// TIA Portal project "CEPS-输送线" (V14)

(* hardware
DEVICE "S7-1200 station_1"  S7-1200 Station
   slot 0: "Rack_0"  S7-1200 Rack  Rack  V1.0
   slot 1: "CEPS传输线"  CPU 1214C DC/DC/DC  6ES7 214-1AG40-0XB0  V4.2
   slot 2: "DI 16x24VDC/DQ 16xRelay_1"  SM 1223 DI16/DQ16 x relay  6ES7 223-1PL32-0XB0  V2.0
   slot 3: "AQ 2x14BIT_1"  SM 1232 AQ2  6ES7 232-4HB32-0XB0  V2.0
DEVICE "HMI"  KTP900 Basic PN
   slot 0: "KTP900 Basic PN"  KTP900 Basic PN  6AV2 123-2JB03-0AX0  14.0.1.0
   slot 1: "HMI_RT_2"  KTP900 Basic PN  6AV2 123-2JB03-0AX0  14.0.1.0
   slot 5: "HMI.IE_CP_1"  PROFINET Interface  14.0.1.0
      slot 1: "PROFINET Interface_1"  PROFINET Interface
         slot 1: "Port_1"  Port
*)

// ===== PLC "CEPS传输线"  CPU 1214C DC/DC/DC =====

VAR_GLOBAL   // PLC tag table "默认变量表"
   "前/后急停按钮" AT %I0.0 : Bool;
   "前/后启动按钮" AT %I0.1 : Bool;
   "前输送线电机变频器报警" AT %I0.2 : Bool;
   "后输送线电机变频器报警" AT %I0.3 : Bool;
   "后方下轨道进料口有料检测" AT %I0.4 : Bool;
   "后升降台有料检测" AT %I0.5 : Bool;
   "前方下轨道出料口有料检测" AT %I0.6 : Bool;
   "前升降台有料检测" AT %I0.7 : Bool;
   "备用2" AT %I1.0 : Bool;
   "前升降台升到位" AT %I1.1 : Bool;
   "前升降台降到位" AT %I1.2 : Bool;
   "后升降台升到位" AT %I1.3 : Bool;
   "后升降台降到位" AT %I1.4 : Bool;
   "备用1" AT %I1.5 : Bool;
   "工位1放行按钮" AT %I2.0 : Bool;
   "工位2放行按钮" AT %I2.1 : Bool;
   "工位3放行按钮" AT %I2.2 : Bool;
   "工位4放行按钮" AT %I2.3 : Bool;
   "工位5放行按钮" AT %I2.4 : Bool;
   "工位6放行按钮" AT %I2.5 : Bool;
   "工位7放行按钮" AT %I2.6 : Bool;
   "前升降台上轨道进料口料盘有料防呆检测" AT %I2.7 : Bool;
   "工位1光电检测" AT %I3.0 : Bool;
   "工位2光电检测" AT %I3.1 : Bool;
   "工位3光电检测" AT %I3.2 : Bool;
   "工位4光电检测" AT %I3.3 : Bool;
   "工位5光电检测" AT %I3.4 : Bool;
   "工位6光电检测" AT %I3.5 : Bool;
   "工位7光电检测" AT %I3.6 : Bool;
   "备用3" AT %I3.7 : Bool;
   "前输送电机启动" AT %Q0.0 : Bool;
   "前输送电机故障复位" AT %Q0.1 : Bool;
   "后输送电机启动" AT %Q0.2 : Bool;
   "后输送电机故障复位" AT %Q0.3 : Bool;
   "前升降台电机正转" AT %Q0.4 : Bool;
   "前升降台电机反转" AT %Q0.5 : Bool;
   "后升降台电机正转" AT %Q0.6 : Bool;
   "后升降台电机反转" AT %Q0.7 : Bool;
   "总气源控制" AT %Q1.0 : Bool;
   "工位3阻挡气缸上升" AT %Q1.1 : Bool;
   "工位1阻挡气缸下降" AT %Q2.0 : Bool;
   "工位2阻挡气缸下降" AT %Q2.1 : Bool;
   "工位3阻挡气缸下降" AT %Q2.2 : Bool;
   "工位4阻挡气缸下降" AT %Q2.3 : Bool;
   "工位5阻挡气缸下降" AT %Q2.4 : Bool;
   "工位6阻挡气缸下降" AT %Q2.5 : Bool;
   "工位7阻挡气缸下降" AT %Q2.6 : Bool;
   "后方下轨道进料口阻挡气缸下降" AT %Q2.7 : Bool;
   "前升降气缸上升" AT %Q3.0 : Bool;
   "前升降气缸下降" AT %Q3.1 : Bool;
   "后升降气缸上升" AT %Q3.2 : Bool;
   "后升降气缸下降" AT %Q3.3 : Bool;
   "后方下轨道阻挡气缸下降" AT %Q3.4 : Bool;
   "后方下轨道阻挡气缸上升" AT %Q3.5 : Bool;
   "工位4阻挡气缸上升" AT %Q3.6 : Bool;
   "工位5阻挡气缸上升" AT %Q3.7 : Bool;
   "System_Byte" AT %MB1 : Byte;
   "FirstScan" AT %M1.0 : Bool;
   "DiagStatusUpdate" AT %M1.1 : Bool;
   "AlwaysTRUE" AT %M1.2 : Bool;
   "AlwaysFALSE" AT %M1.3 : Bool;
   "Clock_Byte" AT %MB0 : Byte;
   "Clock_10Hz" AT %M0.0 : Bool;
   "Clock_5Hz" AT %M0.1 : Bool;
   "Clock_2.5Hz" AT %M0.2 : Bool;
   "Clock_2Hz" AT %M0.3 : Bool;
   "Clock_1.25Hz" AT %M0.4 : Bool;
   "Clock_1Hz" AT %M0.5 : Bool;
   "Clock_0.625Hz" AT %M0.6 : Bool;
   "Clock_0.5Hz" AT %M0.7 : Bool;
   "前输送线电机启动HMI" AT %M10.0 : Bool;
   "前输送线电机停止HMI" AT %M10.1 : Bool;
   "后输送线电机启动HMI" AT %M10.2 : Bool;
   "后输送线电机停止HMI" AT %M10.3 : Bool;
   "前升降台内部电机正转HMI" AT %M10.4 : Bool;
   "前升降台内部电机反转HMI" AT %M10.5 : Bool;
   "前升降台内部电机停止运行HMI" AT %M10.6 : Bool;
   "后升降台内部电机正转HMI" AT %M10.7 : Bool;
   "后升降台内部电机反转HMI" AT %M11.0 : Bool;
   "后升降台内部电机停止运行HMI" AT %M11.1 : Bool;
   "前升降气缸上升HMI" AT %M11.2 : Bool;
   "前升降气缸下降HMI" AT %M11.3 : Bool;
   "后升降气缸上升HMI" AT %M11.4 : Bool;
   "后升降气缸下降HMI" AT %M11.5 : Bool;
   "工位1阻挡气缸上升HMI" AT %M11.6 : Bool;
   "工位1阻挡气缸下降HMI" AT %M11.7 : Bool;
   "工位2阻挡气缸上升HMI" AT %M12.0 : Bool;
   "工位2阻挡气缸下降HMI" AT %M12.1 : Bool;
   "工位3阻挡气缸上升HMI" AT %M12.2 : Bool;
   "工位3阻挡气缸下降HMI" AT %M12.3 : Bool;
   "工位4阻挡气缸上升HMI" AT %M12.4 : Bool;
   "工位4阻挡气缸下降HMI" AT %M12.5 : Bool;
   "工位5阻挡气缸上升HMI" AT %M12.6 : Bool;
   "工位5阻挡气缸下降HMI" AT %M12.7 : Bool;
   "Tag_1" AT %Q4.0 : Bool;
   "工位6阻挡气缸上升HMI" AT %M13.0 : Bool;
   "工位6阻挡气缸下降HMI" AT %M13.1 : Bool;
   "工位7阻挡气缸上升HMI" AT %M13.2 : Bool;
   "工位7阻挡气缸下降HMI" AT %M13.3 : Bool;
   "后方下轨道进料口阻挡气缸上升HMI" AT %M13.4 : Bool;
   "后方下轨道进料口阻挡气缸下降HMI" AT %M13.5 : Bool;
   "后方下轨道阻挡气缸上升HMI" AT %M13.6 : Bool;
   "后方下轨道阻挡气缸下降HMI" AT %M13.7 : Bool;
   "Auto_step" AT %MW50 : Int;
   "Tag_3" AT %MW52 : Int;
   "线体启动HMI" AT %M20.0 : Bool;
   "P0" AT %M4000.0 : Bool;
   "P1" AT %M4000.1 : Bool;
   "P2" AT %M4000.2 : Bool;
   "P3" AT %M4000.3 : Bool;
   "P4" AT %M4000.4 : Bool;
   "P5" AT %M4000.5 : Bool;
   "P6" AT %M4000.6 : Bool;
   "P7" AT %M4000.7 : Bool;
   "P8" AT %M4001.0 : Bool;
   "P9" AT %M4001.1 : Bool;
   "P10" AT %M4001.2 : Bool;
   "P11" AT %M4001.3 : Bool;
   "P12" AT %M4001.4 : Bool;
   "P13" AT %M4001.5 : Bool;
   "P14" AT %M4001.6 : Bool;
   "P15" AT %M4001.7 : Bool;
   "P16" AT %M4002.0 : Bool;
   "P17" AT %M4002.1 : Bool;
   "P18" AT %M4002.2 : Bool;
   "P19" AT %M4002.3 : Bool;
   "P20" AT %M4002.4 : Bool;
   "P21" AT %M4002.5 : Bool;
   "P22" AT %M4002.6 : Bool;
   "P23" AT %M4002.7 : Bool;
   "P24" AT %M4003.0 : Bool;
   "P25" AT %M4003.1 : Bool;
   "P26" AT %M4003.2 : Bool;
   "P27" AT %M4003.3 : Bool;
   "P28" AT %M4003.4 : Bool;
   "P29" AT %M4003.5 : Bool;
   "P30" AT %M4003.6 : Bool;
   "P31" AT %M4003.7 : Bool;
   "P32" AT %M4004.0 : Bool;
   "P33" AT %M4004.1 : Bool;
   "P34" AT %M4004.2 : Bool;
   "P35" AT %M4004.3 : Bool;
   "P36" AT %M4004.4 : Bool;
   "P37" AT %M4004.5 : Bool;
   "P38" AT %M4004.6 : Bool;
   "P39" AT %M4004.7 : Bool;
   "P40" AT %M4005.0 : Bool;
   "P41" AT %M4005.1 : Bool;
   "P42" AT %M4005.2 : Bool;
   "P43" AT %M4005.3 : Bool;
   "P44" AT %M4005.4 : Bool;
   "P45" AT %M4005.5 : Bool;
   "P46" AT %M4005.6 : Bool;
   "P47" AT %M4005.7 : Bool;
   "P48" AT %M4006.0 : Bool;
   "P49" AT %M4006.1 : Bool;
   "P50" AT %M4006.2 : Bool;
   "P51" AT %M4006.3 : Bool;
   "P52" AT %M4006.4 : Bool;
   "P53" AT %M4006.5 : Bool;
   "P54" AT %M4006.6 : Bool;
   "P55" AT %M4006.7 : Bool;
   "P56" AT %M4007.0 : Bool;
   "P57" AT %M4007.1 : Bool;
   "P58" AT %M4007.2 : Bool;
   "P59" AT %M4007.3 : Bool;
   "P60" AT %M4007.4 : Bool;
   "P61" AT %M4007.5 : Bool;
   "P62" AT %M4007.6 : Bool;
   "P63" AT %M4007.7 : Bool;
   "P64" AT %M4008.0 : Bool;
   "P65" AT %M4008.1 : Bool;
   "P66" AT %M4008.2 : Bool;
   "P67" AT %M4008.3 : Bool;
   "P68" AT %M4008.4 : Bool;
   "P69" AT %M4008.5 : Bool;
   "P70" AT %M4008.6 : Bool;
   "P71" AT %M4008.7 : Bool;
   "P72" AT %M4009.0 : Bool;
   "P73" AT %M4009.1 : Bool;
   "P74" AT %M4009.2 : Bool;
   "P75" AT %M4009.3 : Bool;
   "P76" AT %M4009.4 : Bool;
   "P77" AT %M4009.5 : Bool;
   "P78" AT %M4009.6 : Bool;
   "P79" AT %M4009.7 : Bool;
   "P80" AT %M4010.0 : Bool;
   "P81" AT %M4010.1 : Bool;
   "P82" AT %M4010.2 : Bool;
   "P83" AT %M4010.3 : Bool;
   "P84" AT %M4010.4 : Bool;
   "P85" AT %M4010.5 : Bool;
   "P86" AT %M4010.6 : Bool;
   "P87" AT %M4010.7 : Bool;
   "P88" AT %M4011.0 : Bool;
   "P89" AT %M4011.1 : Bool;
   "P90" AT %M4011.2 : Bool;
   "P91" AT %M4011.3 : Bool;
   "P92" AT %M4011.4 : Bool;
   "P93" AT %M4011.5 : Bool;
   "P94" AT %M4011.6 : Bool;
   "P95" AT %M4011.7 : Bool;
   "P96" AT %M4012.0 : Bool;
   "P97" AT %M4012.1 : Bool;
   "P98" AT %M4012.2 : Bool;
   "P99" AT %M4012.3 : Bool;
   "P100" AT %M4012.4 : Bool;
   "线体停止HMI" AT %M20.1 : Bool;
   "前升降台皮带电机正在工作" AT %M100.0 : Bool;
   "后升降台皮带电机正在工作" AT %M100.1 : Bool;
   "前升降台皮带电机显示到HMI状态号" AT %MW2000 : Word;
   "Tag_2" AT %QW112 : Int;
   "Tag_4" AT %QW114 : Int;
   "后升降台皮带电机显示到HMI状态号" AT %MW2002 : Int;
   "前输送线电机显示到HMI状态号" AT %MW2004 : Int;
   "后输送线电机显示到HMI状态号" AT %MW2006 : Int;
   "故障复位HMI" AT %M20.2 : Bool;
   "前升降气缸上升超时报警" AT %M1000.0 : Bool;
   "前升降气缸下降超时报警" AT %M1000.1 : Bool;
   "报警1" AT %MW1000 : Int;
   "后升降气缸上升超时报警" AT %M1000.2 : Bool;
   "后升降气缸下降超时报警" AT %M1000.3 : Bool;
   "前输送电机变频器故障报警" AT %M1000.4 : Bool;
   "后输送电机变频器故障报警" AT %M1000.5 : Bool;
   "急停按下报警" AT %M1000.6 : Bool;
   "设备状态号" AT %MW54 : Int;
   "工位7按钮已按下，待工件流入前升降台，禁止工位7按钮触发" AT %M100.2 : Bool;
   "放行判断" AT %M100.3 : Bool;
END_VAR

DATA_BLOCK "MB_TCON"   // DB1
{ S7_Optimized_Access := 'TRUE' }
VERSION : 0.1
   VAR
      MB_TCON : TCON_IP_v4;
   END_VAR
BEGIN
   MB_TCON.InterfaceId := 64;
   MB_TCON.ID := 1;
   MB_TCON.LocalPort := 502;
END_DATA_BLOCK

DATA_BLOCK "保持数据块"   // DB23
{ S7_Optimized_Access := 'FALSE' }
VERSION : 0.1
   VAR
      产品型号 : Int;
      前输送电机变频器设定频率 : Int;
      后输送电机变频器设定频率 : Int;
      "手动放行/自动放行" : Bool;
      滑移力检测工位 : Int;
      上柱管轴承压装工位 : Int;
      拉轴工位 : Int;
      手柄装配工位 : Int;
      上下柱管压装工位 : Int;
      滑移力复测工位 : Int;
      手柄调节机构工位 : Int;
   END_VAR
BEGIN
END_DATA_BLOCK

DATA_BLOCK "MB_DATA"   // DB100
{ S7_Optimized_Access := 'FALSE' }
VERSION : 0.1
   VAR
      设备编号 : Int := 0;
      产品型号 : Int := 0;
      设备状态 : Int;
      错误代码 : Int := 0;
      当前曲线 : Int := 0;
      工位1状态 : Int := 0;
      工位2状态 : Int;
      工位3状态 : Int;
      工位1生产结果 : Int;
      工位2生产结果 : Int;
      工位3生产结果 : Int;
      备用_1 : Int;
      备用_2 : Int;
      备用_3 : Int;
      备用_4 : Int;
      备用_5 : Int;
      复测拉压力传感器 : Array[0..4] of Real;
      复测位移传感器 : Array[0..4] of Real;
      拉轴拉压力传感器 : Array[0..4] of Real;
      传感器4 : Array[0..4] of Real;
      传感器5 : Array[0..4] of Real;
      传感器6 : Array[0..4] of Real;
      传感器7 : Array[0..4] of Real;
      传感器8 : Array[0..4] of Real;
      传感器9 : Array[0..4] of Real;
      传感器10 : Array[0..4] of Real;
      传感器11 : Array[0..4] of Real;
      传感器12 : Array[0..4] of Real;
      传感器13 : Array[0..4] of Real;
      传感器14 : Array[0..4] of Real;
   END_VAR
BEGIN
   复测拉压力传感器[0] := 0.0;   // 压力值
   复测拉压力传感器[1] := 0.0;
   复测位移传感器[0] := 0.0;   // 位移值
   复测位移传感器[1] := 0.0;
   拉轴拉压力传感器[0] := 0.0;   // 压力值
   拉轴拉压力传感器[1] := 0.0;
   复测拉压力传感器[2] := 0.0;
   复测拉压力传感器[3] := 0.0;
   复测拉压力传感器[4] := 0.0;
   复测位移传感器[2] := 0.0;
   复测位移传感器[3] := 0.0;
   复测位移传感器[4] := 0.0;
   拉轴拉压力传感器[2] := 0.0;
   拉轴拉压力传感器[3] := 0.0;
   拉轴拉压力传感器[4] := 0.0;
   传感器6[0] := 0.0;   // 输入轴角度
   传感器6[1] := 0.0;   // 输出轴角度
   传感器6[2] := 0.0;   // 流量
   传感器6[3] := 0.0;   // 输入轴位移
   传感器6[4] := 0.0;
   传感器4[0] := 0.0;   // 量程下限
   传感器4[1] := 200.0;   // 量程上限
   传感器4[2] := 0.0;   // 原始值
   传感器4[3] := 0.0;   // 偏移值
   传感器4[4] := 0.0;   // 标定值
   传感器5[4] := 0.0;   // 标定值
   传感器5[3] := 0.0;   // 偏移值
   传感器5[2] := 0.0;   // 原始值
   传感器5[1] := 2.5;   // 量程上限
   传感器5[0] := 0.0;   // 量程下限
   传感器8[4] := 65.0;   // 温度上限
   传感器8[3] := 35.0;   // 温度下限
   // 传感器9[0] : 接近距离
   // 传感器9[1] : 接近速度
   // 传感器9[2] : 套入距离
   // 传感器9[3] : 套入速度
   // 传感器10[1] : 摆动角度
   // 传感器10[2] : 摆动速度
   // 传感器10[0] : 状态
   // 传感器10[3] : 保护扭矩
   // 传感器12[0] : 速度
   // 传感器12[1] : 换向扭矩
   // 传感器8[0] : 系统流量
   // 传感器8[1] : 试验流量
   // 传感器8[2] : 试验压力
   // 传感器7[0] : 输入轴角度下限
   // 传感器7[1] : 输入轴角度上限
   // 传感器7[2] : 输出轴角度下限
   // 传感器7[3] : 输出轴角度上限
   // 传感器7[4] : 总圈数
   // 传感器13[0] : 内泄露时间
   // 传感器11[0] : 状态
   // 传感器11[1] : 摆动角度
   // 传感器11[2] : 摆动速度
   // 传感器11[3] : 保护扭矩
   // 传感器14[0] : 输入轴速度
END_DATA_BLOCK

// folder: System blocks/Program resources

DATA_BLOCK "IEC_Timer_0_DB"   // DB3
{ S7_Optimized_Access := 'TRUE' }
AUTHOR : Simatic
FAMILY : IEC
NAME : IEC_TMR
VERSION : 1.0
// stored: InstanceOfName IEC_TIMER
"IEC_TIMER"
BEGIN
END_DATA_BLOCK

DATA_BLOCK "IEC_Timer_0_DB_0"   // DB4
{ S7_Optimized_Access := 'TRUE' }
AUTHOR : Simatic
FAMILY : IEC
NAME : IEC_TMR
VERSION : 1.0
// stored: InstanceOfName IEC_TIMER
"IEC_TIMER"
BEGIN
END_DATA_BLOCK

DATA_BLOCK "IEC_Timer_0_DB_1"   // DB5
{ S7_Optimized_Access := 'TRUE' }
AUTHOR : Simatic
FAMILY : IEC
NAME : IEC_TMR
VERSION : 1.0
// stored: InstanceOfName IEC_TIMER
"IEC_TIMER"
BEGIN
END_DATA_BLOCK

DATA_BLOCK "IEC_Timer_0_DB_2"   // DB6
{ S7_Optimized_Access := 'TRUE' }
AUTHOR : Simatic
FAMILY : IEC
NAME : IEC_TMR
VERSION : 1.0
// stored: InstanceOfName IEC_TIMER
"IEC_TIMER"
BEGIN
END_DATA_BLOCK

DATA_BLOCK "IEC_Timer_0_DB_3"   // DB7
{ S7_Optimized_Access := 'TRUE' }
AUTHOR : Simatic
FAMILY : IEC
NAME : IEC_TMR
VERSION : 1.0
// stored: InstanceOfName IEC_TIMER
"IEC_TIMER"
BEGIN
END_DATA_BLOCK

DATA_BLOCK "IEC_Timer_0_DB_4"   // DB8
{ S7_Optimized_Access := 'TRUE' }
AUTHOR : Simatic
FAMILY : IEC
NAME : IEC_TMR
VERSION : 1.0
// stored: InstanceOfName IEC_TIMER
"IEC_TIMER"
BEGIN
END_DATA_BLOCK

DATA_BLOCK "IEC_Timer_0_DB_5"   // DB9
{ S7_Optimized_Access := 'TRUE' }
AUTHOR : Simatic
FAMILY : IEC
NAME : IEC_TMR
VERSION : 1.0
// stored: InstanceOfName IEC_TIMER
"IEC_TIMER"
BEGIN
END_DATA_BLOCK

DATA_BLOCK "IEC_Timer_0_DB_6"   // DB10
{ S7_Optimized_Access := 'TRUE' }
AUTHOR : Simatic
FAMILY : IEC
NAME : IEC_TMR
VERSION : 1.0
// stored: InstanceOfName IEC_TIMER
"IEC_TIMER"
BEGIN
END_DATA_BLOCK

DATA_BLOCK "IEC_Timer_0_DB_7"   // DB11
{ S7_Optimized_Access := 'TRUE' }
AUTHOR : Simatic
FAMILY : IEC
NAME : IEC_TMR
VERSION : 1.0
// stored: InstanceOfName IEC_TIMER
"IEC_TIMER"
BEGIN
END_DATA_BLOCK

DATA_BLOCK "IEC_Timer_0_DB_8"   // DB12
{ S7_Optimized_Access := 'TRUE' }
AUTHOR : Simatic
FAMILY : IEC
NAME : IEC_TMR
VERSION : 1.0
// stored: InstanceOfName IEC_TIMER
"IEC_TIMER"
BEGIN
END_DATA_BLOCK

DATA_BLOCK "IEC_Timer_0_DB_9"   // DB13
{ S7_Optimized_Access := 'TRUE' }
AUTHOR : Simatic
FAMILY : IEC
NAME : IEC_TMR
VERSION : 1.0
// stored: InstanceOfName IEC_TIMER
"IEC_TIMER"
BEGIN
END_DATA_BLOCK

DATA_BLOCK "IEC_Timer_0_DB_10"   // DB14
{ S7_Optimized_Access := 'TRUE' }
AUTHOR : Simatic
FAMILY : IEC
NAME : IEC_TMR
VERSION : 1.0
// stored: InstanceOfName IEC_TIMER
"IEC_TIMER"
BEGIN
END_DATA_BLOCK

DATA_BLOCK "IEC_Timer_0_DB_11"   // DB15
{ S7_Optimized_Access := 'TRUE' }
AUTHOR : Simatic
FAMILY : IEC
NAME : IEC_TMR
VERSION : 1.0
// stored: InstanceOfName IEC_TIMER
"IEC_TIMER"
BEGIN
END_DATA_BLOCK

DATA_BLOCK "IEC_Timer_0_DB_12"   // DB16
{ S7_Optimized_Access := 'TRUE' }
AUTHOR : Simatic
FAMILY : IEC
NAME : IEC_TMR
VERSION : 1.0
// stored: InstanceOfName IEC_TIMER
"IEC_TIMER"
BEGIN
END_DATA_BLOCK

DATA_BLOCK "IEC_Timer_0_DB_13"   // DB17
{ S7_Optimized_Access := 'TRUE' }
AUTHOR : Simatic
FAMILY : IEC
NAME : IEC_TMR
VERSION : 1.0
// stored: InstanceOfName IEC_TIMER
"IEC_TIMER"
BEGIN
END_DATA_BLOCK

DATA_BLOCK "IEC_Timer_0_DB_14"   // DB18
{ S7_Optimized_Access := 'TRUE' }
AUTHOR : Simatic
FAMILY : IEC
NAME : IEC_TMR
VERSION : 1.0
// stored: InstanceOfName IEC_TIMER
"IEC_TIMER"
BEGIN
END_DATA_BLOCK

DATA_BLOCK "IEC_Timer_0_DB_15"   // DB19
{ S7_Optimized_Access := 'TRUE' }
AUTHOR : Simatic
FAMILY : IEC
NAME : IEC_TMR
VERSION : 1.0
// stored: InstanceOfName IEC_TIMER
"IEC_TIMER"
BEGIN
END_DATA_BLOCK

DATA_BLOCK "IEC_Timer_0_DB_16"   // DB20
{ S7_Optimized_Access := 'TRUE' }
AUTHOR : Simatic
FAMILY : IEC
NAME : IEC_TMR
VERSION : 1.0
// stored: InstanceOfName IEC_TIMER
"IEC_TIMER"
BEGIN
END_DATA_BLOCK

DATA_BLOCK "IEC_Timer_0_DB_17"   // DB21
{ S7_Optimized_Access := 'TRUE' }
AUTHOR : Simatic
FAMILY : IEC
NAME : IEC_TMR
VERSION : 1.0
// stored: InstanceOfName IEC_TIMER
"IEC_TIMER"
BEGIN
END_DATA_BLOCK

DATA_BLOCK "IEC_Timer_0_DB_18"   // DB22
{ S7_Optimized_Access := 'TRUE' }
AUTHOR : Simatic
FAMILY : IEC
NAME : IEC_TMR
VERSION : 1.0
// stored: InstanceOfName IEC_TIMER
"IEC_TIMER"
BEGIN
END_DATA_BLOCK

DATA_BLOCK "IEC_Timer_0_DB_19"   // DB24
{ S7_Optimized_Access := 'TRUE' }
AUTHOR : Simatic
FAMILY : IEC
NAME : IEC_TMR
VERSION : 1.0
// stored: InstanceOfName IEC_TIMER
"IEC_TIMER"
BEGIN
END_DATA_BLOCK

DATA_BLOCK "IEC_Timer_0_DB_20"   // DB25
{ S7_Optimized_Access := 'TRUE' }
AUTHOR : Simatic
FAMILY : IEC
NAME : IEC_TMR
VERSION : 1.0
// stored: InstanceOfName IEC_TIMER
"IEC_TIMER"
BEGIN
END_DATA_BLOCK

DATA_BLOCK "IEC_Timer_0_DB_21"   // DB26
{ S7_Optimized_Access := 'TRUE' }
AUTHOR : Simatic
FAMILY : IEC
NAME : IEC_TMR
VERSION : 1.0
// stored: InstanceOfName IEC_TIMER
"IEC_TIMER"
BEGIN
END_DATA_BLOCK

DATA_BLOCK "IEC_Timer_0_DB_22"   // DB27
{ S7_Optimized_Access := 'TRUE' }
AUTHOR : Simatic
FAMILY : IEC
NAME : IEC_TMR
VERSION : 1.0
// stored: InstanceOfName IEC_TIMER
"IEC_TIMER"
BEGIN
END_DATA_BLOCK

DATA_BLOCK "IEC_Timer_0_DB_23"   // DB28
{ S7_Optimized_Access := 'TRUE' }
AUTHOR : Simatic
FAMILY : IEC
NAME : IEC_TMR
VERSION : 1.0
// stored: InstanceOfName IEC_TIMER
"IEC_TIMER"
BEGIN
END_DATA_BLOCK

DATA_BLOCK "IEC_Timer_0_DB_24"   // DB29
{ S7_Optimized_Access := 'TRUE' }
AUTHOR : Simatic
FAMILY : IEC
NAME : IEC_TMR
VERSION : 1.0
// stored: InstanceOfName IEC_TIMER
"IEC_TIMER"
BEGIN
END_DATA_BLOCK

DATA_BLOCK "IEC_Timer_0_DB_25"   // DB30
{ S7_Optimized_Access := 'TRUE' }
AUTHOR : Simatic
FAMILY : IEC
NAME : IEC_TMR
VERSION : 1.0
// stored: InstanceOfName IEC_TIMER
"IEC_TIMER"
BEGIN
END_DATA_BLOCK

DATA_BLOCK "IEC_Timer_0_DB_26"   // DB31
{ S7_Optimized_Access := 'TRUE' }
AUTHOR : Simatic
FAMILY : IEC
NAME : IEC_TMR
VERSION : 1.0
// stored: InstanceOfName IEC_TIMER
"IEC_TIMER"
BEGIN
END_DATA_BLOCK

DATA_BLOCK "IEC_Timer_0_DB_27"   // DB32
{ S7_Optimized_Access := 'TRUE' }
AUTHOR : Simatic
FAMILY : IEC
NAME : IEC_TMR
VERSION : 1.0
// stored: InstanceOfName IEC_TIMER
"IEC_TIMER"
BEGIN
END_DATA_BLOCK

DATA_BLOCK "IEC_Timer_0_DB_28"   // DB33
{ S7_Optimized_Access := 'TRUE' }
AUTHOR : Simatic
FAMILY : IEC
NAME : IEC_TMR
VERSION : 1.0
// stored: InstanceOfName IEC_TIMER
"IEC_TIMER"
BEGIN
END_DATA_BLOCK

DATA_BLOCK "IEC_Timer_0_DB_29"   // DB34
{ S7_Optimized_Access := 'TRUE' }
AUTHOR : Simatic
FAMILY : IEC
NAME : IEC_TMR
VERSION : 1.0
// stored: InstanceOfName IEC_TIMER
"IEC_TIMER"
BEGIN
END_DATA_BLOCK

DATA_BLOCK "IEC_Timer_0_DB_30"   // DB35
{ S7_Optimized_Access := 'TRUE' }
AUTHOR : Simatic
FAMILY : IEC
NAME : IEC_TMR
VERSION : 1.0
// stored: InstanceOfName IEC_TIMER
"IEC_TIMER"
BEGIN
END_DATA_BLOCK

// folder: (top level)

FUNCTION "手动程序" : Void   // FC1, LAD
{ S7_Optimized_Access := 'TRUE' }
VERSION : 0.1
   VAR_TEMP   // added for the SCL form of the ladder/FBD networks
      _w1 : Bool;
      _w2 : Bool;
   END_VAR
BEGIN

REGION Network 1: 前输送线电机控制
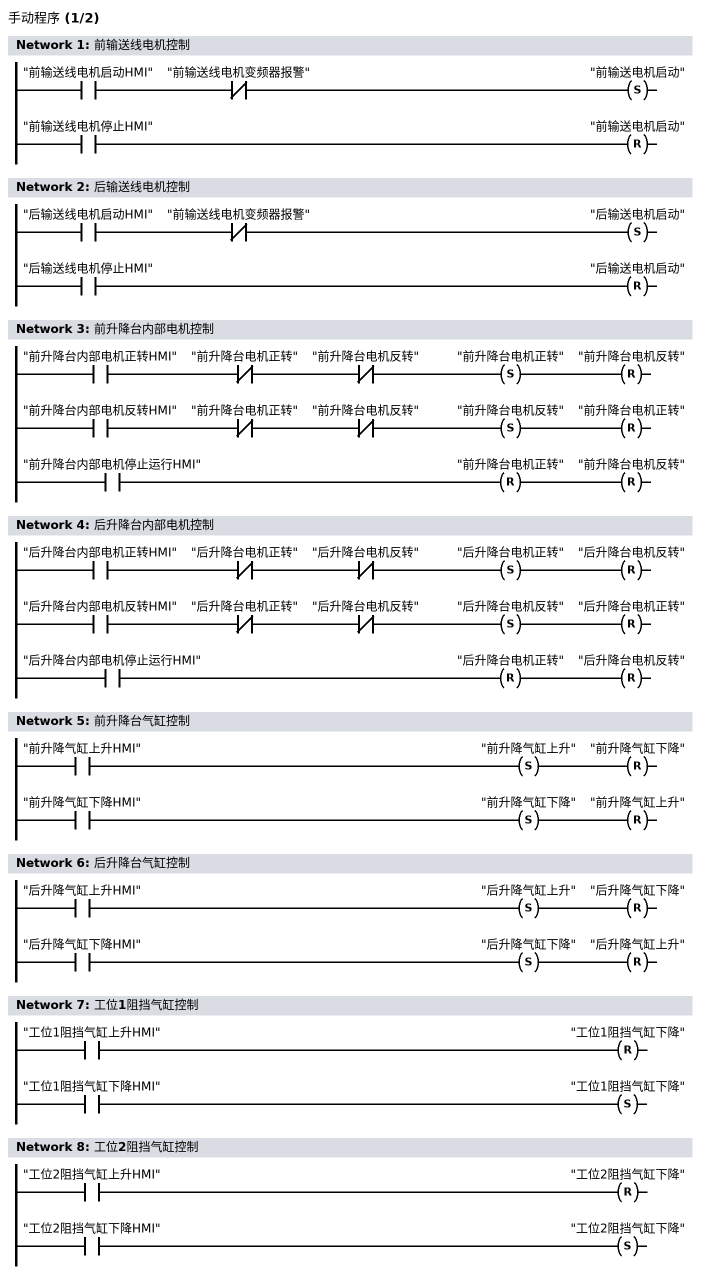
   RUNG wire#powerrail
      Contact( "前输送线电机启动HMI" )
      I_Contact( "前输送线电机变频器报警" )
      S_Coil( "前输送电机启动" )
   END_RUNG
   RUNG wire#powerrail
      Contact( "前输送线电机停止HMI" )
      R_Coil( "前输送电机启动" )
   END_RUNG
   // the same network as SCL:
   IF "前输送线电机启动HMI" AND NOT "前输送线电机变频器报警" THEN "前输送电机启动" := TRUE; END_IF;
   IF "前输送线电机停止HMI" THEN "前输送电机启动" := FALSE; END_IF;
END_REGION

REGION Network 2: 后输送线电机控制
   RUNG wire#powerrail
      Contact( "后输送线电机启动HMI" )
      I_Contact( "前输送线电机变频器报警" )
      S_Coil( "后输送电机启动" )
   END_RUNG
   RUNG wire#powerrail
      Contact( "后输送线电机停止HMI" )
      R_Coil( "后输送电机启动" )
   END_RUNG
   // the same network as SCL:
   IF "后输送线电机启动HMI" AND NOT "前输送线电机变频器报警" THEN "后输送电机启动" := TRUE; END_IF;
   IF "后输送线电机停止HMI" THEN "后输送电机启动" := FALSE; END_IF;
END_REGION

REGION Network 3: 前升降台内部电机控制
   RUNG wire#powerrail
      Contact( "前升降台内部电机正转HMI" )
      I_Contact( "前升降台电机正转" )
      I_Contact( "前升降台电机反转" )
      S_Coil( "前升降台电机正转" )
      R_Coil( "前升降台电机反转" )
   END_RUNG
   RUNG wire#powerrail
      Contact( "前升降台内部电机反转HMI" )
      I_Contact( "前升降台电机正转" )
      I_Contact( "前升降台电机反转" )
      S_Coil( "前升降台电机反转" )
      R_Coil( "前升降台电机正转" )
   END_RUNG
   RUNG wire#powerrail
      Contact( "前升降台内部电机停止运行HMI" )
      R_Coil( "前升降台电机正转" )
      R_Coil( "前升降台电机反转" )
   END_RUNG
   // the same network as SCL:
   #_w1 := "前升降台内部电机正转HMI" AND NOT "前升降台电机正转" AND NOT "前升降台电机反转";
   IF #_w1 THEN
       "前升降台电机正转" := TRUE;
       "前升降台电机反转" := FALSE;
   END_IF;
   #_w2 := "前升降台内部电机反转HMI" AND NOT "前升降台电机正转" AND NOT "前升降台电机反转";
   IF #_w2 THEN
       "前升降台电机反转" := TRUE;
       "前升降台电机正转" := FALSE;
   END_IF;
   IF "前升降台内部电机停止运行HMI" THEN
       "前升降台电机正转" := FALSE;
       "前升降台电机反转" := FALSE;
   END_IF;
END_REGION

REGION Network 4: 后升降台内部电机控制
   RUNG wire#powerrail
      Contact( "后升降台内部电机正转HMI" )
      I_Contact( "后升降台电机正转" )
      I_Contact( "后升降台电机反转" )
      S_Coil( "后升降台电机正转" )
      R_Coil( "后升降台电机反转" )
   END_RUNG
   RUNG wire#powerrail
      Contact( "后升降台内部电机反转HMI" )
      I_Contact( "后升降台电机正转" )
      I_Contact( "后升降台电机反转" )
      S_Coil( "后升降台电机反转" )
      R_Coil( "后升降台电机正转" )
   END_RUNG
   RUNG wire#powerrail
      Contact( "后升降台内部电机停止运行HMI" )
      R_Coil( "后升降台电机正转" )
      R_Coil( "后升降台电机反转" )
   END_RUNG
   // the same network as SCL:
   #_w1 := "后升降台内部电机正转HMI" AND NOT "后升降台电机正转" AND NOT "后升降台电机反转";
   IF #_w1 THEN
       "后升降台电机正转" := TRUE;
       "后升降台电机反转" := FALSE;
   END_IF;
   #_w2 := "后升降台内部电机反转HMI" AND NOT "后升降台电机正转" AND NOT "后升降台电机反转";
   IF #_w2 THEN
       "后升降台电机反转" := TRUE;
       "后升降台电机正转" := FALSE;
   END_IF;
   IF "后升降台内部电机停止运行HMI" THEN
       "后升降台电机正转" := FALSE;
       "后升降台电机反转" := FALSE;
   END_IF;
END_REGION

REGION Network 5: 前升降台气缸控制
   RUNG wire#powerrail
      Contact( "前升降气缸上升HMI" )
      S_Coil( "前升降气缸上升" )
      R_Coil( "前升降气缸下降" )
   END_RUNG
   RUNG wire#powerrail
      Contact( "前升降气缸下降HMI" )
      S_Coil( "前升降气缸下降" )
      R_Coil( "前升降气缸上升" )
   END_RUNG
   // the same network as SCL:
   IF "前升降气缸上升HMI" THEN
       "前升降气缸上升" := TRUE;
       "前升降气缸下降" := FALSE;
   END_IF;
   IF "前升降气缸下降HMI" THEN
       "前升降气缸下降" := TRUE;
       "前升降气缸上升" := FALSE;
   END_IF;
END_REGION

REGION Network 6: 后升降台气缸控制
   RUNG wire#powerrail
      Contact( "后升降气缸上升HMI" )
      S_Coil( "后升降气缸上升" )
      R_Coil( "后升降气缸下降" )
   END_RUNG
   RUNG wire#powerrail
      Contact( "后升降气缸下降HMI" )
      S_Coil( "后升降气缸下降" )
      R_Coil( "后升降气缸上升" )
   END_RUNG
   // the same network as SCL:
   IF "后升降气缸上升HMI" THEN
       "后升降气缸上升" := TRUE;
       "后升降气缸下降" := FALSE;
   END_IF;
   IF "后升降气缸下降HMI" THEN
       "后升降气缸下降" := TRUE;
       "后升降气缸上升" := FALSE;
   END_IF;
END_REGION

REGION Network 7: 工位1阻挡气缸控制
   RUNG wire#powerrail
      Contact( "工位1阻挡气缸上升HMI" )
      R_Coil( "工位1阻挡气缸下降" )
   END_RUNG
   RUNG wire#powerrail
      Contact( "工位1阻挡气缸下降HMI" )
      S_Coil( "工位1阻挡气缸下降" )
   END_RUNG
   // the same network as SCL:
   IF "工位1阻挡气缸上升HMI" THEN "工位1阻挡气缸下降" := FALSE; END_IF;
   IF "工位1阻挡气缸下降HMI" THEN "工位1阻挡气缸下降" := TRUE; END_IF;
END_REGION

REGION Network 8: 工位2阻挡气缸控制
   RUNG wire#powerrail
      Contact( "工位2阻挡气缸上升HMI" )
      R_Coil( "工位2阻挡气缸下降" )
   END_RUNG
   RUNG wire#powerrail
      Contact( "工位2阻挡气缸下降HMI" )
      S_Coil( "工位2阻挡气缸下降" )
   END_RUNG
   // the same network as SCL:
   IF "工位2阻挡气缸上升HMI" THEN "工位2阻挡气缸下降" := FALSE; END_IF;
   IF "工位2阻挡气缸下降HMI" THEN "工位2阻挡气缸下降" := TRUE; END_IF;
END_REGION

REGION Network 9: 工位3阻挡气缸控制
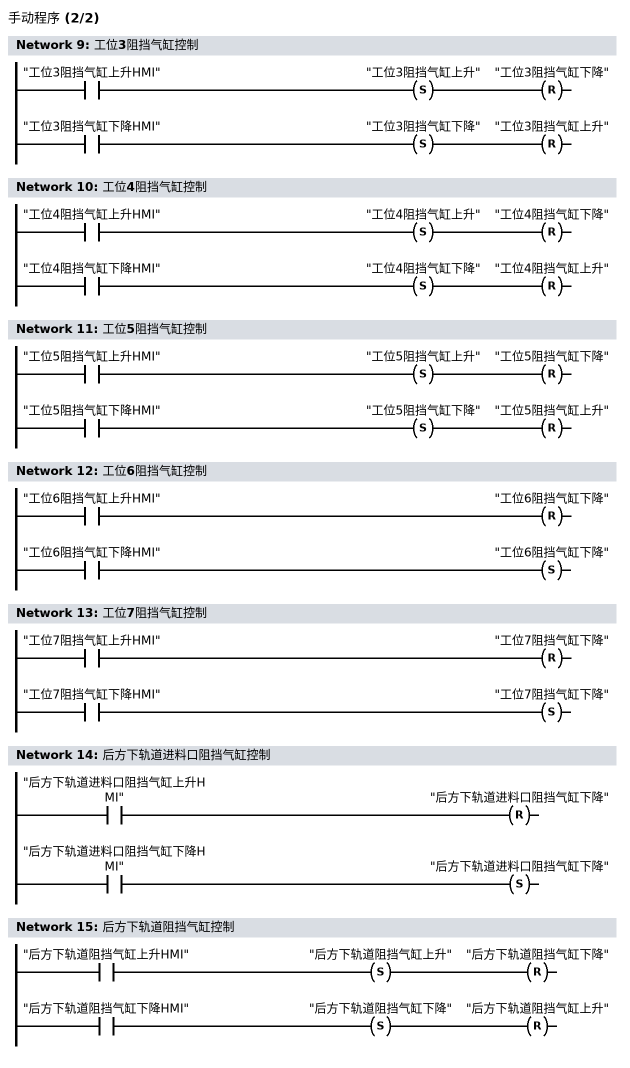
   RUNG wire#powerrail
      Contact( "工位3阻挡气缸上升HMI" )
      S_Coil( "工位3阻挡气缸上升" )
      R_Coil( "工位3阻挡气缸下降" )
   END_RUNG
   RUNG wire#powerrail
      Contact( "工位3阻挡气缸下降HMI" )
      S_Coil( "工位3阻挡气缸下降" )
      R_Coil( "工位3阻挡气缸上升" )
   END_RUNG
   // the same network as SCL:
   IF "工位3阻挡气缸上升HMI" THEN
       "工位3阻挡气缸上升" := TRUE;
       "工位3阻挡气缸下降" := FALSE;
   END_IF;
   IF "工位3阻挡气缸下降HMI" THEN
       "工位3阻挡气缸下降" := TRUE;
       "工位3阻挡气缸上升" := FALSE;
   END_IF;
END_REGION

REGION Network 10: 工位4阻挡气缸控制
   RUNG wire#powerrail
      Contact( "工位4阻挡气缸上升HMI" )
      S_Coil( "工位4阻挡气缸上升" )
      R_Coil( "工位4阻挡气缸下降" )
   END_RUNG
   RUNG wire#powerrail
      Contact( "工位4阻挡气缸下降HMI" )
      S_Coil( "工位4阻挡气缸下降" )
      R_Coil( "工位4阻挡气缸上升" )
   END_RUNG
   // the same network as SCL:
   IF "工位4阻挡气缸上升HMI" THEN
       "工位4阻挡气缸上升" := TRUE;
       "工位4阻挡气缸下降" := FALSE;
   END_IF;
   IF "工位4阻挡气缸下降HMI" THEN
       "工位4阻挡气缸下降" := TRUE;
       "工位4阻挡气缸上升" := FALSE;
   END_IF;
END_REGION

REGION Network 11: 工位5阻挡气缸控制
   RUNG wire#powerrail
      Contact( "工位5阻挡气缸上升HMI" )
      S_Coil( "工位5阻挡气缸上升" )
      R_Coil( "工位5阻挡气缸下降" )
   END_RUNG
   RUNG wire#powerrail
      Contact( "工位5阻挡气缸下降HMI" )
      S_Coil( "工位5阻挡气缸下降" )
      R_Coil( "工位5阻挡气缸上升" )
   END_RUNG
   // the same network as SCL:
   IF "工位5阻挡气缸上升HMI" THEN
       "工位5阻挡气缸上升" := TRUE;
       "工位5阻挡气缸下降" := FALSE;
   END_IF;
   IF "工位5阻挡气缸下降HMI" THEN
       "工位5阻挡气缸下降" := TRUE;
       "工位5阻挡气缸上升" := FALSE;
   END_IF;
END_REGION

REGION Network 12: 工位6阻挡气缸控制
   RUNG wire#powerrail
      Contact( "工位6阻挡气缸上升HMI" )
      R_Coil( "工位6阻挡气缸下降" )
   END_RUNG
   RUNG wire#powerrail
      Contact( "工位6阻挡气缸下降HMI" )
      S_Coil( "工位6阻挡气缸下降" )
   END_RUNG
   // the same network as SCL:
   IF "工位6阻挡气缸上升HMI" THEN "工位6阻挡气缸下降" := FALSE; END_IF;
   IF "工位6阻挡气缸下降HMI" THEN "工位6阻挡气缸下降" := TRUE; END_IF;
END_REGION

REGION Network 13: 工位7阻挡气缸控制
   RUNG wire#powerrail
      Contact( "工位7阻挡气缸上升HMI" )
      R_Coil( "工位7阻挡气缸下降" )
   END_RUNG
   RUNG wire#powerrail
      Contact( "工位7阻挡气缸下降HMI" )
      S_Coil( "工位7阻挡气缸下降" )
   END_RUNG
   // the same network as SCL:
   IF "工位7阻挡气缸上升HMI" THEN "工位7阻挡气缸下降" := FALSE; END_IF;
   IF "工位7阻挡气缸下降HMI" THEN "工位7阻挡气缸下降" := TRUE; END_IF;
END_REGION

REGION Network 14: 后方下轨道进料口阻挡气缸控制
   RUNG wire#powerrail
      Contact( "后方下轨道进料口阻挡气缸上升HMI" )
      R_Coil( "后方下轨道进料口阻挡气缸下降" )
   END_RUNG
   RUNG wire#powerrail
      Contact( "后方下轨道进料口阻挡气缸下降HMI" )
      S_Coil( "后方下轨道进料口阻挡气缸下降" )
   END_RUNG
   // the same network as SCL:
   IF "后方下轨道进料口阻挡气缸上升HMI" THEN "后方下轨道进料口阻挡气缸下降" := FALSE; END_IF;
   IF "后方下轨道进料口阻挡气缸下降HMI" THEN "后方下轨道进料口阻挡气缸下降" := TRUE; END_IF;
END_REGION

REGION Network 15: 后方下轨道阻挡气缸控制
   RUNG wire#powerrail
      Contact( "后方下轨道阻挡气缸上升HMI" )
      S_Coil( "后方下轨道阻挡气缸上升" )
      R_Coil( "后方下轨道阻挡气缸下降" )
   END_RUNG
   RUNG wire#powerrail
      Contact( "后方下轨道阻挡气缸下降HMI" )
      S_Coil( "后方下轨道阻挡气缸下降" )
      R_Coil( "后方下轨道阻挡气缸上升" )
   END_RUNG
   // the same network as SCL:
   IF "后方下轨道阻挡气缸上升HMI" THEN
       "后方下轨道阻挡气缸上升" := TRUE;
       "后方下轨道阻挡气缸下降" := FALSE;
   END_IF;
   IF "后方下轨道阻挡气缸下降HMI" THEN
       "后方下轨道阻挡气缸下降" := TRUE;
       "后方下轨道阻挡气缸上升" := FALSE;
   END_IF;
END_REGION
END_FUNCTION

FUNCTION "模拟量" : Void   // FC2, LAD
{ S7_Optimized_Access := 'TRUE' }
VERSION : 0.1
   VAR_TEMP
      前变频器比例存储 : Real;
      后变频器比例存储 : Real;
   END_VAR
BEGIN

REGION Network 1
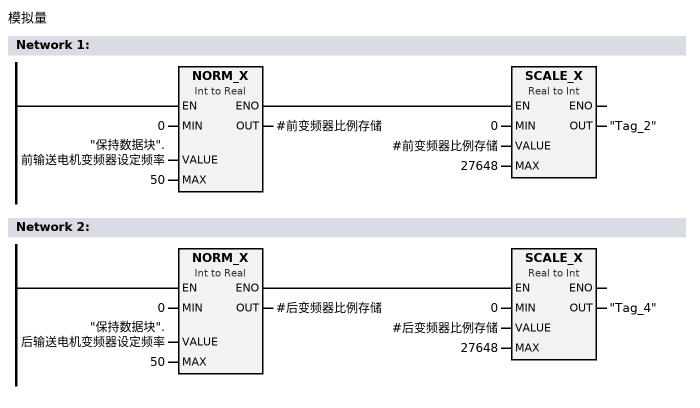
   RUNG wire#powerrail
      { S7_Templates := "[SrcType := Int, DestType := Real]" } Normalize(min := 0, value := "保持数据块".前输送电机变频器设定频率, max := 50, out => #前变频器比例存储)
      { S7_Templates := "[SrcType := Real, DestType := Int]" } Scale(min := 0, value := #前变频器比例存储, max := 27648, out => "Tag_2")
   END_RUNG
   // the same network as SCL:
   #前变频器比例存储 := NORM_X(MIN := 0, VALUE := "保持数据块".前输送电机变频器设定频率, MAX := 50);
   "Tag_2" := SCALE_X(MIN := 0, VALUE := #前变频器比例存储, MAX := 27648);
END_REGION

REGION Network 2
   RUNG wire#powerrail
      { S7_Templates := "[SrcType := Int, DestType := Real]" } Normalize(min := 0, value := "保持数据块".后输送电机变频器设定频率, max := 50, out => #后变频器比例存储)
      { S7_Templates := "[SrcType := Real, DestType := Int]" } Scale(min := 0, value := #后变频器比例存储, max := 27648, out => "Tag_4")
   END_RUNG
   // the same network as SCL:
   #后变频器比例存储 := NORM_X(MIN := 0, VALUE := "保持数据块".后输送电机变频器设定频率, MAX := 50);
   "Tag_4" := SCALE_X(MIN := 0, VALUE := #后变频器比例存储, MAX := 27648);
END_REGION
END_FUNCTION

FUNCTION "自动程序" : Void   // FC3, LAD
{ S7_Optimized_Access := 'TRUE' }
VERSION : 0.1
   VAR_TEMP   // added for the SCL form of the ladder/FBD networks
      _w1 : Bool;
      _w2 : Bool;
      _w3 : Bool;
      _w4 : Bool;
      _w5 : Bool;
      _w6 : Bool;
      _w7 : Bool;
      _w8 : Bool;
   END_VAR
BEGIN

REGION Network 1: 启动按下：线体阻挡气缸全部下降
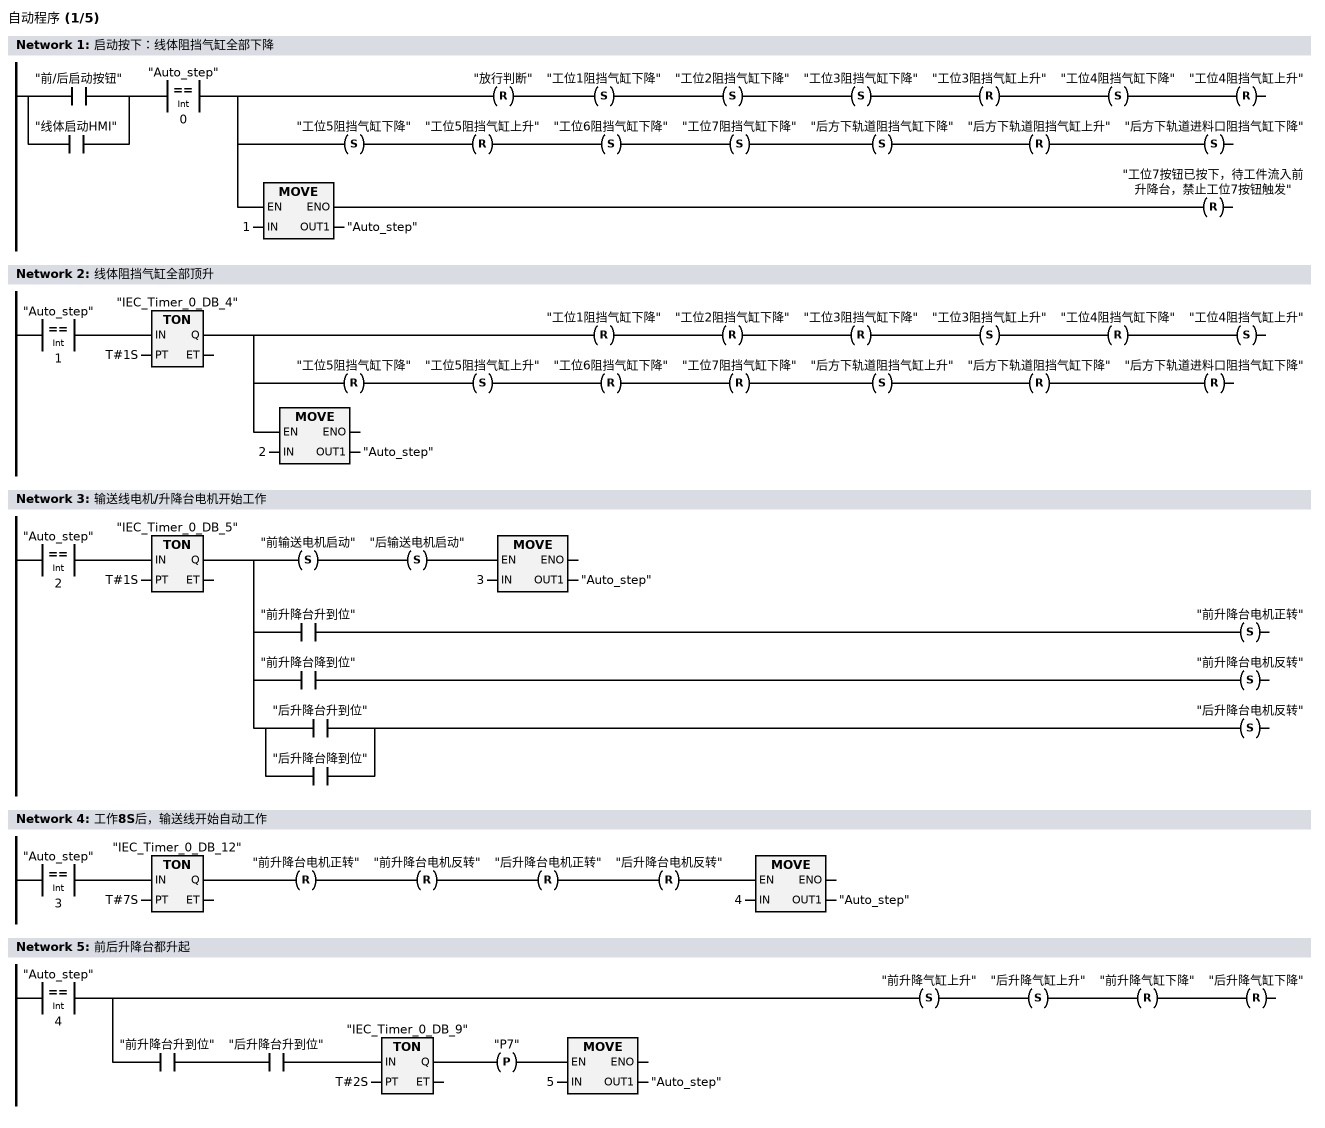
   RUNG wire#powerrail
      Contact( "前/后启动按钮" )
      wire#w1
      { S7_Templates := "SrcType := Int" } EQ_Contact(in1 := "Auto_step", in2 := 0)
      wire#w2
      R_Coil( "放行判断" )
      S_Coil( "工位1阻挡气缸下降" )
      S_Coil( "工位2阻挡气缸下降" )
      S_Coil( "工位3阻挡气缸下降" )
      R_Coil( "工位3阻挡气缸上升" )
      S_Coil( "工位4阻挡气缸下降" )
      R_Coil( "工位4阻挡气缸上升" )
   END_RUNG
   RUNG wire#powerrail
      Contact( "线体启动HMI" )
   END_RUNG wire#w1
   RUNG wire#w2
      S_Coil( "工位5阻挡气缸下降" )
      R_Coil( "工位5阻挡气缸上升" )
      S_Coil( "工位6阻挡气缸下降" )
      S_Coil( "工位7阻挡气缸下降" )
      S_Coil( "后方下轨道阻挡气缸下降" )
      R_Coil( "后方下轨道阻挡气缸上升" )
      S_Coil( "后方下轨道进料口阻挡气缸下降" )
   END_RUNG
   RUNG wire#w2
      Move(in := 1, out1 => "Auto_step")
      R_Coil( "工位7按钮已按下，待工件流入前升降台，禁止工位7按钮触发" )
   END_RUNG
   // the same network as SCL:
   IF ("前/后启动按钮" OR "线体启动HMI") AND ("Auto_step" = 0) THEN
       "放行判断" := FALSE;
       "工位1阻挡气缸下降" := TRUE;
       "工位2阻挡气缸下降" := TRUE;
       "工位3阻挡气缸下降" := TRUE;
       "工位3阻挡气缸上升" := FALSE;
       "工位4阻挡气缸下降" := TRUE;
       "工位4阻挡气缸上升" := FALSE;
       "工位5阻挡气缸下降" := TRUE;
       "工位5阻挡气缸上升" := FALSE;
       "工位6阻挡气缸下降" := TRUE;
       "工位7阻挡气缸下降" := TRUE;
       "后方下轨道阻挡气缸下降" := TRUE;
       "后方下轨道阻挡气缸上升" := FALSE;
       "后方下轨道进料口阻挡气缸下降" := TRUE;
   END_IF;
   #_w1 := ("前/后启动按钮" OR "线体启动HMI") AND ("Auto_step" = 0);
   IF #_w1 THEN
       "Auto_step" := 1;
       "工位7按钮已按下，待工件流入前升降台，禁止工位7按钮触发" := FALSE;
   END_IF;
END_REGION

REGION Network 2: 线体阻挡气缸全部顶升
   "IEC_Timer_0_DB_4".TON(IN := "Auto_step" = 1, PT := T#1S);
   IF "IEC_Timer_0_DB_4".Q THEN
       "工位1阻挡气缸下降" := FALSE;
       "工位2阻挡气缸下降" := FALSE;
       "工位3阻挡气缸下降" := FALSE;
       "工位3阻挡气缸上升" := TRUE;
       "工位4阻挡气缸下降" := FALSE;
       "工位4阻挡气缸上升" := TRUE;
       "工位5阻挡气缸下降" := FALSE;
       "工位5阻挡气缸上升" := TRUE;
       "工位6阻挡气缸下降" := FALSE;
       "工位7阻挡气缸下降" := FALSE;
       "后方下轨道阻挡气缸上升" := TRUE;
       "后方下轨道阻挡气缸下降" := FALSE;
       "后方下轨道进料口阻挡气缸下降" := FALSE;
       "Auto_step" := 2;
   END_IF;
END_REGION

REGION Network 3: 输送线电机/升降台电机开始工作
   "IEC_Timer_0_DB_5".TON(IN := "Auto_step" = 2, PT := T#1S);
   IF "IEC_Timer_0_DB_5".Q THEN
       "前输送电机启动" := TRUE;
       "后输送电机启动" := TRUE;
       "Auto_step" := 3;
   END_IF;
   IF "IEC_Timer_0_DB_5".Q AND "前升降台升到位" THEN "前升降台电机正转" := TRUE; END_IF;
   IF "IEC_Timer_0_DB_5".Q AND "前升降台降到位" THEN "前升降台电机反转" := TRUE; END_IF;
   IF "IEC_Timer_0_DB_5".Q AND ("后升降台升到位" OR "后升降台降到位") THEN "后升降台电机反转" := TRUE; END_IF;
END_REGION

REGION Network 4: 工作8S后，输送线开始自动工作
   "IEC_Timer_0_DB_12".TON(IN := "Auto_step" = 3, PT := T#7S);
   IF "IEC_Timer_0_DB_12".Q THEN
       "前升降台电机正转" := FALSE;
       "前升降台电机反转" := FALSE;
       "后升降台电机正转" := FALSE;
       "后升降台电机反转" := FALSE;
       "Auto_step" := 4;
   END_IF;
END_REGION

REGION Network 5: 前后升降台都升起
   #_w1 := "Auto_step" = 4;
   IF #_w1 THEN
       "前升降气缸上升" := TRUE;
       "后升降气缸上升" := TRUE;
       "前升降气缸下降" := FALSE;
       "后升降气缸下降" := FALSE;
   END_IF;
   "IEC_Timer_0_DB_9".TON(IN := #_w1 AND "前升降台升到位" AND "后升降台升到位", PT := T#2S);
   #_w2 := "IEC_Timer_0_DB_9".Q AND NOT "P7";   // rising edge
   "P7" := "IEC_Timer_0_DB_9".Q;
   IF #_w2 THEN "Auto_step" := 5; END_IF;
END_REGION

REGION Network 6: 工位1
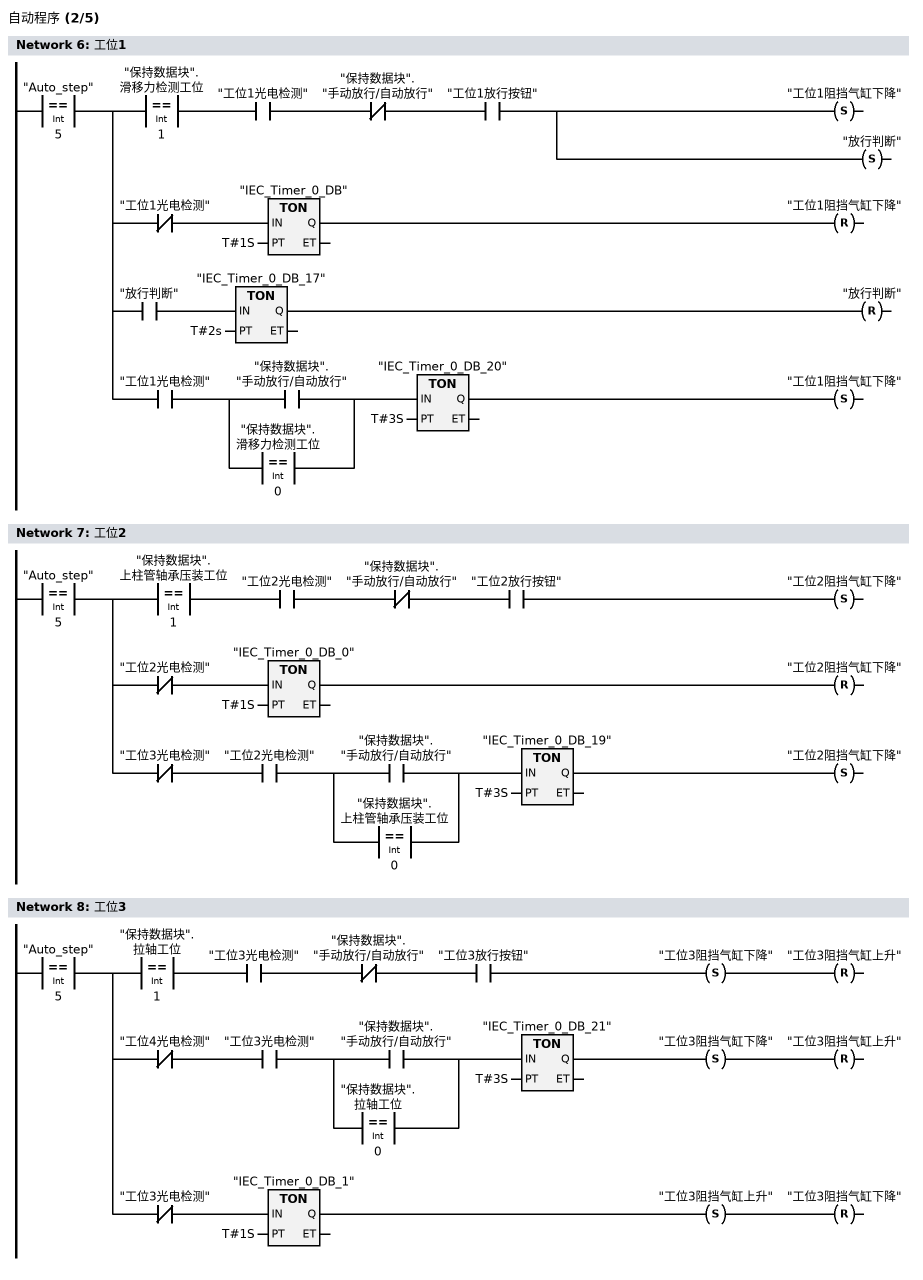
   #_w1 := "Auto_step" = 5;
   IF #_w1 AND ("保持数据块".滑移力检测工位 = 1) AND "工位1光电检测" AND NOT "保持数据块"."手动放行/自动放行" AND "工位1放行按钮" THEN
       "工位1阻挡气缸下降" := TRUE;
       "放行判断" := TRUE;
   END_IF;
   "IEC_Timer_0_DB".TON(IN := #_w1 AND NOT "工位1光电检测", PT := T#1S);
   IF "IEC_Timer_0_DB".Q THEN "工位1阻挡气缸下降" := FALSE; END_IF;
   "IEC_Timer_0_DB_17".TON(IN := #_w1 AND "放行判断", PT := T#2s);
   IF "IEC_Timer_0_DB_17".Q THEN "放行判断" := FALSE; END_IF;
   "IEC_Timer_0_DB_20".TON(IN := #_w1 AND "工位1光电检测" AND ("保持数据块"."手动放行/自动放行" OR ("保持数据块".滑移力检测工位 = 0)),
                           PT := T#3S);
   IF "IEC_Timer_0_DB_20".Q THEN "工位1阻挡气缸下降" := TRUE; END_IF;
END_REGION

REGION Network 7: 工位2
   #_w1 := "Auto_step" = 5;
   IF #_w1 AND ("保持数据块".上柱管轴承压装工位 = 1) AND "工位2光电检测" AND NOT "保持数据块"."手动放行/自动放行" AND "工位2放行按钮" THEN
       "工位2阻挡气缸下降" := TRUE;
   END_IF;
   "IEC_Timer_0_DB_0".TON(IN := #_w1 AND NOT "工位2光电检测", PT := T#1S);
   IF "IEC_Timer_0_DB_0".Q THEN "工位2阻挡气缸下降" := FALSE; END_IF;
   "IEC_Timer_0_DB_19".TON(IN := #_w1 AND NOT "工位3光电检测" AND "工位2光电检测" AND ("保持数据块"."手动放行/自动放行" OR ("保持数据块".上柱管轴承压装工位 = 0)),
                           PT := T#3S);
   IF "IEC_Timer_0_DB_19".Q THEN "工位2阻挡气缸下降" := TRUE; END_IF;
END_REGION

REGION Network 8: 工位3
   #_w1 := "Auto_step" = 5;
   IF #_w1 AND ("保持数据块".拉轴工位 = 1) AND "工位3光电检测" AND NOT "保持数据块"."手动放行/自动放行" AND "工位3放行按钮" THEN
       "工位3阻挡气缸下降" := TRUE;
       "工位3阻挡气缸上升" := FALSE;
   END_IF;
   "IEC_Timer_0_DB_21".TON(IN := #_w1 AND NOT "工位4光电检测" AND "工位3光电检测" AND ("保持数据块"."手动放行/自动放行" OR ("保持数据块".拉轴工位 = 0)),
                           PT := T#3S);
   IF "IEC_Timer_0_DB_21".Q THEN
       "工位3阻挡气缸下降" := TRUE;
       "工位3阻挡气缸上升" := FALSE;
   END_IF;
   "IEC_Timer_0_DB_1".TON(IN := #_w1 AND NOT "工位3光电检测", PT := T#1S);
   IF "IEC_Timer_0_DB_1".Q THEN
       "工位3阻挡气缸上升" := TRUE;
       "工位3阻挡气缸下降" := FALSE;
   END_IF;
END_REGION

REGION Network 9: 工位4
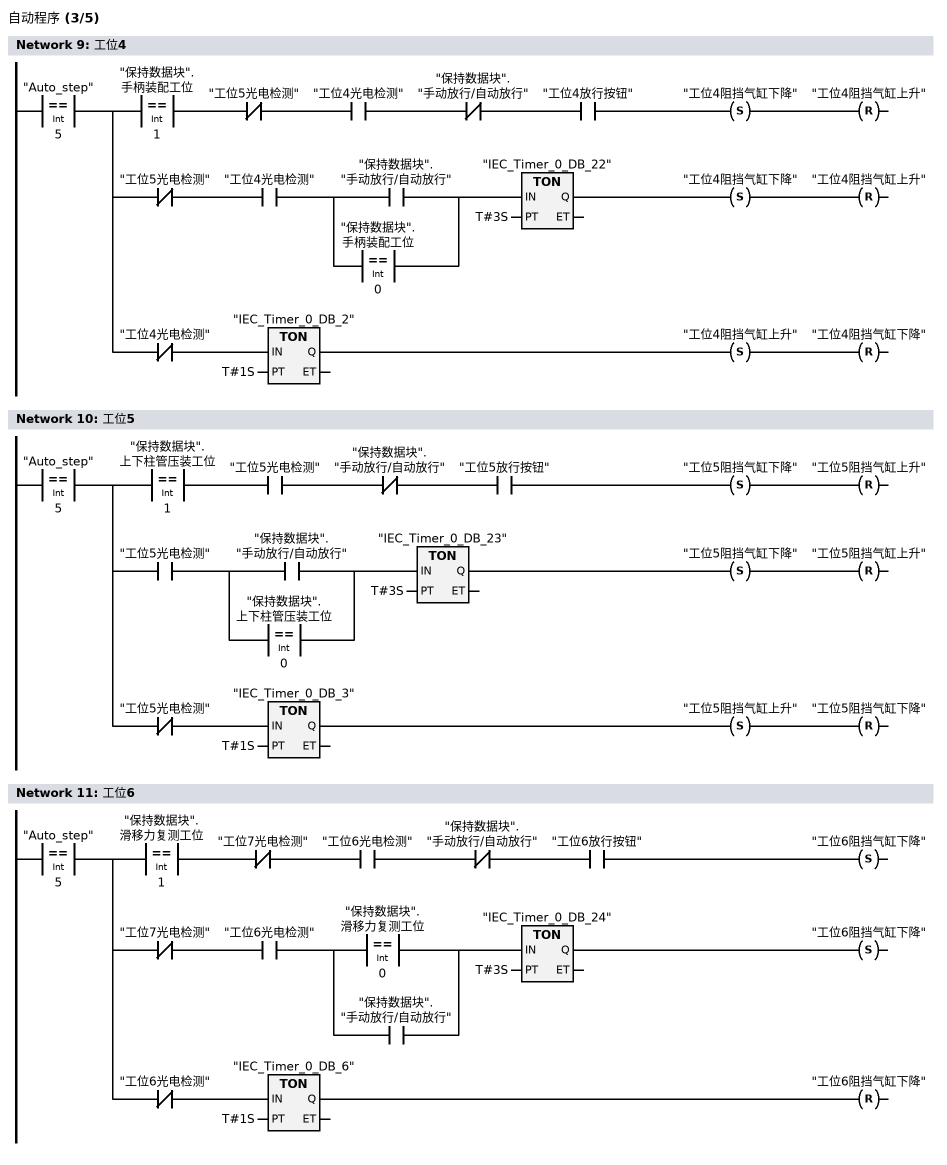
   #_w1 := "Auto_step" = 5;
   IF #_w1 AND ("保持数据块".手柄装配工位 = 1) AND NOT "工位5光电检测" AND "工位4光电检测" AND NOT "保持数据块"."手动放行/自动放行" AND "工位4放行按钮" THEN
       "工位4阻挡气缸下降" := TRUE;
       "工位4阻挡气缸上升" := FALSE;
   END_IF;
   "IEC_Timer_0_DB_22".TON(IN := #_w1 AND NOT "工位5光电检测" AND "工位4光电检测" AND ("保持数据块"."手动放行/自动放行" OR ("保持数据块".手柄装配工位 = 0)),
                           PT := T#3S);
   IF "IEC_Timer_0_DB_22".Q THEN
       "工位4阻挡气缸下降" := TRUE;
       "工位4阻挡气缸上升" := FALSE;
   END_IF;
   "IEC_Timer_0_DB_2".TON(IN := #_w1 AND NOT "工位4光电检测", PT := T#1S);
   IF "IEC_Timer_0_DB_2".Q THEN
       "工位4阻挡气缸上升" := TRUE;
       "工位4阻挡气缸下降" := FALSE;
   END_IF;
END_REGION

REGION Network 10: 工位5
   #_w1 := "Auto_step" = 5;
   IF #_w1 AND ("保持数据块".上下柱管压装工位 = 1) AND "工位5光电检测" AND NOT "保持数据块"."手动放行/自动放行" AND "工位5放行按钮" THEN
       "工位5阻挡气缸下降" := TRUE;
       "工位5阻挡气缸上升" := FALSE;
   END_IF;
   "IEC_Timer_0_DB_23".TON(IN := #_w1 AND "工位5光电检测" AND ("保持数据块"."手动放行/自动放行" OR ("保持数据块".上下柱管压装工位 = 0)),
                           PT := T#3S);
   IF "IEC_Timer_0_DB_23".Q THEN
       "工位5阻挡气缸下降" := TRUE;
       "工位5阻挡气缸上升" := FALSE;
   END_IF;
   "IEC_Timer_0_DB_3".TON(IN := #_w1 AND NOT "工位5光电检测", PT := T#1S);
   IF "IEC_Timer_0_DB_3".Q THEN
       "工位5阻挡气缸上升" := TRUE;
       "工位5阻挡气缸下降" := FALSE;
   END_IF;
END_REGION

REGION Network 11: 工位6
   #_w1 := "Auto_step" = 5;
   IF #_w1 AND ("保持数据块".滑移力复测工位 = 1) AND NOT "工位7光电检测" AND "工位6光电检测" AND NOT "保持数据块"."手动放行/自动放行" AND "工位6放行按钮" THEN
       "工位6阻挡气缸下降" := TRUE;
   END_IF;
   "IEC_Timer_0_DB_24".TON(IN := #_w1 AND NOT "工位7光电检测" AND "工位6光电检测" AND (("保持数据块".滑移力复测工位 = 0) OR "保持数据块"."手动放行/自动放行"),
                           PT := T#3S);
   IF "IEC_Timer_0_DB_24".Q THEN "工位6阻挡气缸下降" := TRUE; END_IF;
   "IEC_Timer_0_DB_6".TON(IN := #_w1 AND NOT "工位6光电检测", PT := T#1S);
   IF "IEC_Timer_0_DB_6".Q THEN "工位6阻挡气缸下降" := FALSE; END_IF;
END_REGION

REGION Network 12: 工位7
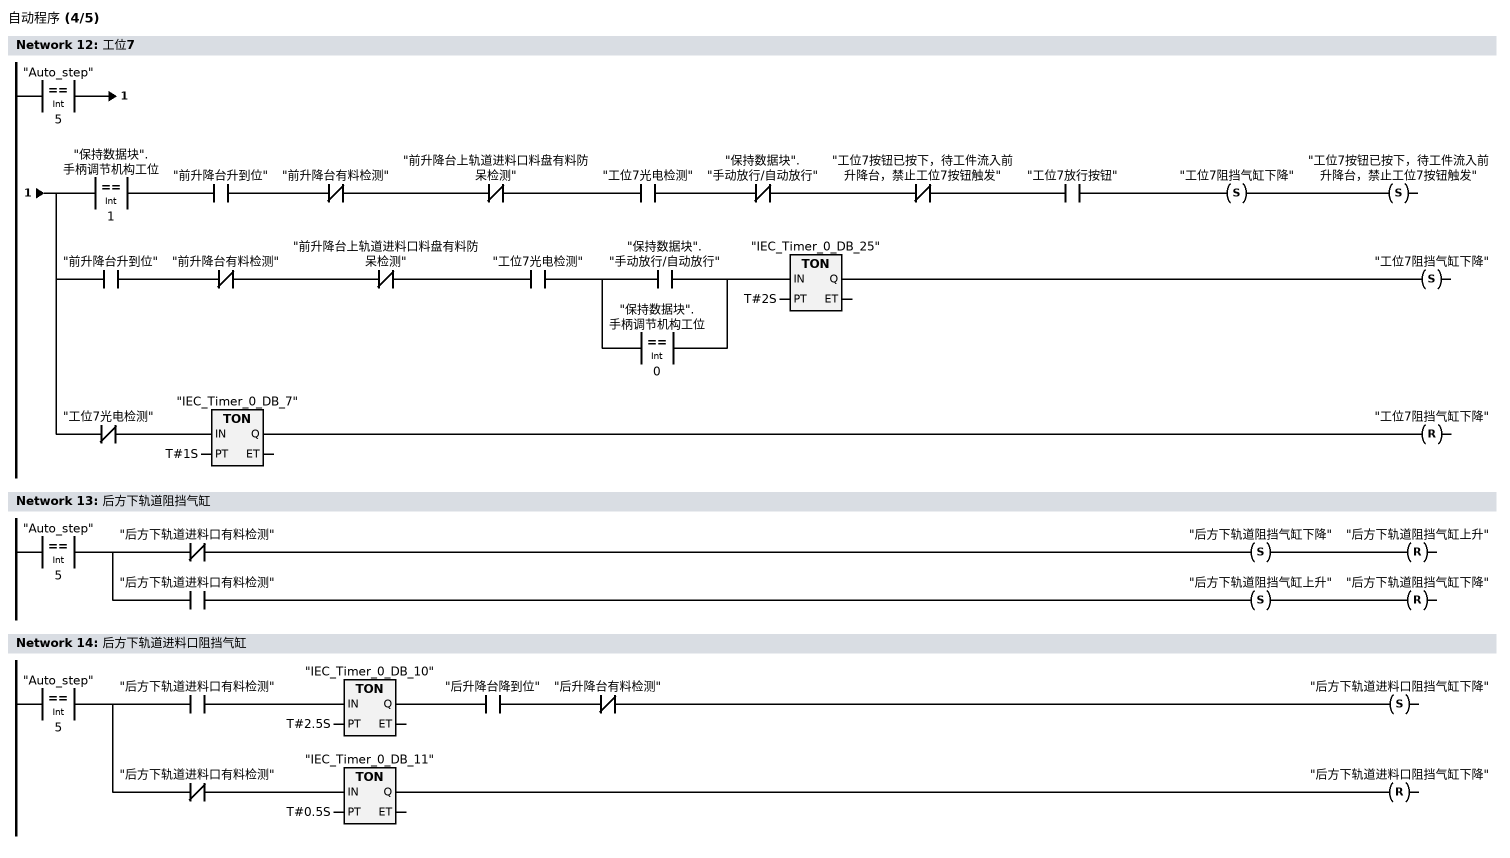
   #_w1 := "Auto_step" = 5;
   IF #_w1 AND ("保持数据块".手柄调节机构工位 = 1) AND "前升降台升到位" AND NOT "前升降台有料检测" AND NOT "前升降台上轨道进料口料盘有料防呆检测" AND "工位7光电检测" AND NOT "保持数据块"."手动放行/自动放行" AND NOT "工位7按钮已按下，待工件流入前升降台，禁止工位7按钮触发" AND "工位7放行按钮" THEN
       "工位7阻挡气缸下降" := TRUE;
       "工位7按钮已按下，待工件流入前升降台，禁止工位7按钮触发" := TRUE;
   END_IF;
   "IEC_Timer_0_DB_25".TON(IN := #_w1 AND "前升降台升到位" AND NOT "前升降台有料检测" AND NOT "前升降台上轨道进料口料盘有料防呆检测" AND "工位7光电检测" AND ("保持数据块"."手动放行/自动放行" OR ("保持数据块".手柄调节机构工位 = 0)),
                           PT := T#2S);
   IF "IEC_Timer_0_DB_25".Q THEN "工位7阻挡气缸下降" := TRUE; END_IF;
   "IEC_Timer_0_DB_7".TON(IN := #_w1 AND NOT "工位7光电检测", PT := T#1S);
   IF "IEC_Timer_0_DB_7".Q THEN "工位7阻挡气缸下降" := FALSE; END_IF;
END_REGION

REGION Network 13: 后方下轨道阻挡气缸
   RUNG wire#powerrail
      { S7_Templates := "SrcType := Int" } EQ_Contact(in1 := "Auto_step", in2 := 5)
      wire#w1
      I_Contact( "后方下轨道进料口有料检测" )
      S_Coil( "后方下轨道阻挡气缸下降" )
      R_Coil( "后方下轨道阻挡气缸上升" )
   END_RUNG
   RUNG wire#w1
      Contact( "后方下轨道进料口有料检测" )
      S_Coil( "后方下轨道阻挡气缸上升" )
      R_Coil( "后方下轨道阻挡气缸下降" )
   END_RUNG
   // the same network as SCL:
   #_w1 := "Auto_step" = 5;
   IF #_w1 AND NOT "后方下轨道进料口有料检测" THEN
       "后方下轨道阻挡气缸下降" := TRUE;
       "后方下轨道阻挡气缸上升" := FALSE;
   END_IF;
   IF #_w1 AND "后方下轨道进料口有料检测" THEN
       "后方下轨道阻挡气缸上升" := TRUE;
       "后方下轨道阻挡气缸下降" := FALSE;
   END_IF;
END_REGION

REGION Network 14: 后方下轨道进料口阻挡气缸
   #_w1 := "Auto_step" = 5;
   "IEC_Timer_0_DB_10".TON(IN := #_w1 AND "后方下轨道进料口有料检测", PT := T#2.5S);
   IF "IEC_Timer_0_DB_10".Q AND "后升降台降到位" AND NOT "后升降台有料检测" THEN "后方下轨道进料口阻挡气缸下降" := TRUE; END_IF;
   "IEC_Timer_0_DB_11".TON(IN := #_w1 AND NOT "后方下轨道进料口有料检测", PT := T#0.5S);
   IF "IEC_Timer_0_DB_11".Q THEN "后方下轨道进料口阻挡气缸下降" := FALSE; END_IF;
END_REGION

REGION Network 15: 前升降台气缸与电机
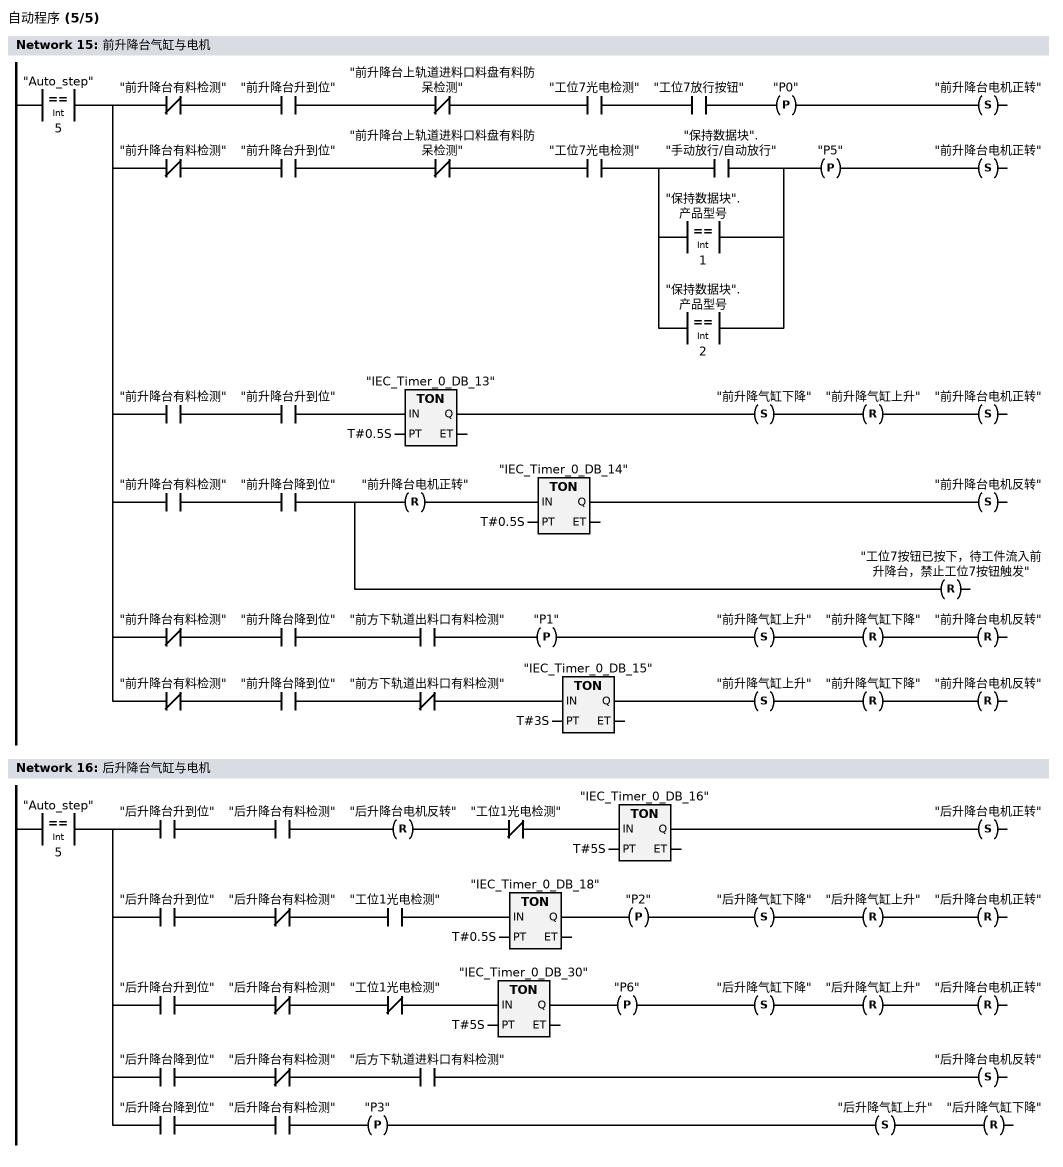
   #_w1 := "Auto_step" = 5;
   #_w2 := #_w1 AND NOT "前升降台有料检测" AND "前升降台升到位" AND NOT "前升降台上轨道进料口料盘有料防呆检测" AND "工位7光电检测" AND "工位7放行按钮";
   #_w3 := #_w2 AND NOT "P0";   // rising edge
   "P0" := #_w2;
   IF #_w3 THEN "前升降台电机正转" := TRUE; END_IF;
   #_w4 := #_w1 AND NOT "前升降台有料检测" AND "前升降台升到位" AND NOT "前升降台上轨道进料口料盘有料防呆检测" AND "工位7光电检测" AND ("保持数据块"."手动放行/自动放行" OR ("保持数据块".产品型号 = 1) OR ("保持数据块".产品型号 = 2));
   #_w5 := #_w4 AND NOT "P5";   // rising edge
   "P5" := #_w4;
   IF #_w5 THEN "前升降台电机正转" := TRUE; END_IF;
   "IEC_Timer_0_DB_13".TON(IN := #_w1 AND "前升降台有料检测" AND "前升降台升到位", PT := T#0.5S);
   IF "IEC_Timer_0_DB_13".Q THEN
       "前升降气缸下降" := TRUE;
       "前升降气缸上升" := FALSE;
       "前升降台电机正转" := TRUE;
   END_IF;
   #_w6 := #_w1 AND "前升降台有料检测" AND "前升降台降到位";
   IF #_w6 THEN "前升降台电机正转" := FALSE; END_IF;
   "IEC_Timer_0_DB_14".TON(IN := #_w6, PT := T#0.5S);
   IF "IEC_Timer_0_DB_14".Q THEN "前升降台电机反转" := TRUE; END_IF;
   IF #_w6 THEN "工位7按钮已按下，待工件流入前升降台，禁止工位7按钮触发" := FALSE; END_IF;
   #_w7 := #_w1 AND NOT "前升降台有料检测" AND "前升降台降到位" AND "前方下轨道出料口有料检测";
   #_w8 := #_w7 AND NOT "P1";   // rising edge
   "P1" := #_w7;
   IF #_w8 THEN
       "前升降气缸上升" := TRUE;
       "前升降气缸下降" := FALSE;
       "前升降台电机反转" := FALSE;
   END_IF;
   "IEC_Timer_0_DB_15".TON(IN := #_w1 AND NOT "前升降台有料检测" AND "前升降台降到位" AND NOT "前方下轨道出料口有料检测", PT := T#3S);
   IF "IEC_Timer_0_DB_15".Q THEN
       "前升降气缸上升" := TRUE;
       "前升降气缸下降" := FALSE;
       "前升降台电机反转" := FALSE;
   END_IF;
END_REGION

REGION Network 16: 后升降台气缸与电机
   #_w1 := "Auto_step" = 5;
   #_w2 := #_w1 AND "后升降台升到位" AND "后升降台有料检测";
   IF #_w2 THEN "后升降台电机反转" := FALSE; END_IF;
   "IEC_Timer_0_DB_16".TON(IN := #_w2 AND NOT "工位1光电检测", PT := T#5S);
   IF "IEC_Timer_0_DB_16".Q THEN "后升降台电机正转" := TRUE; END_IF;
   "IEC_Timer_0_DB_18".TON(IN := #_w1 AND "后升降台升到位" AND NOT "后升降台有料检测" AND "工位1光电检测", PT := T#0.5S);
   #_w3 := "IEC_Timer_0_DB_18".Q AND NOT "P2";   // rising edge
   "P2" := "IEC_Timer_0_DB_18".Q;
   IF #_w3 THEN
       "后升降气缸下降" := TRUE;
       "后升降气缸上升" := FALSE;
       "后升降台电机正转" := FALSE;
   END_IF;
   "IEC_Timer_0_DB_30".TON(IN := #_w1 AND "后升降台升到位" AND NOT "后升降台有料检测" AND NOT "工位1光电检测", PT := T#5S);
   #_w4 := "IEC_Timer_0_DB_30".Q AND NOT "P6";   // rising edge
   "P6" := "IEC_Timer_0_DB_30".Q;
   IF #_w4 THEN
       "后升降气缸下降" := TRUE;
       "后升降气缸上升" := FALSE;
       "后升降台电机正转" := FALSE;
   END_IF;
   IF #_w1 AND "后升降台降到位" AND NOT "后升降台有料检测" AND "后方下轨道进料口有料检测" THEN "后升降台电机反转" := TRUE; END_IF;
   #_w5 := #_w1 AND "后升降台降到位" AND "后升降台有料检测";
   #_w6 := #_w5 AND NOT "P3";   // rising edge
   "P3" := #_w5;
   IF #_w6 THEN
       "后升降气缸上升" := TRUE;
       "后升降气缸下降" := FALSE;
   END_IF;
END_REGION
END_FUNCTION

FUNCTION "PLC/HMI交互" : Void   // FC4, LAD
{ S7_Optimized_Access := 'TRUE' }
VERSION : 0.1
BEGIN

REGION Network 1: 前升降台皮带电机工作状态显示到HMI
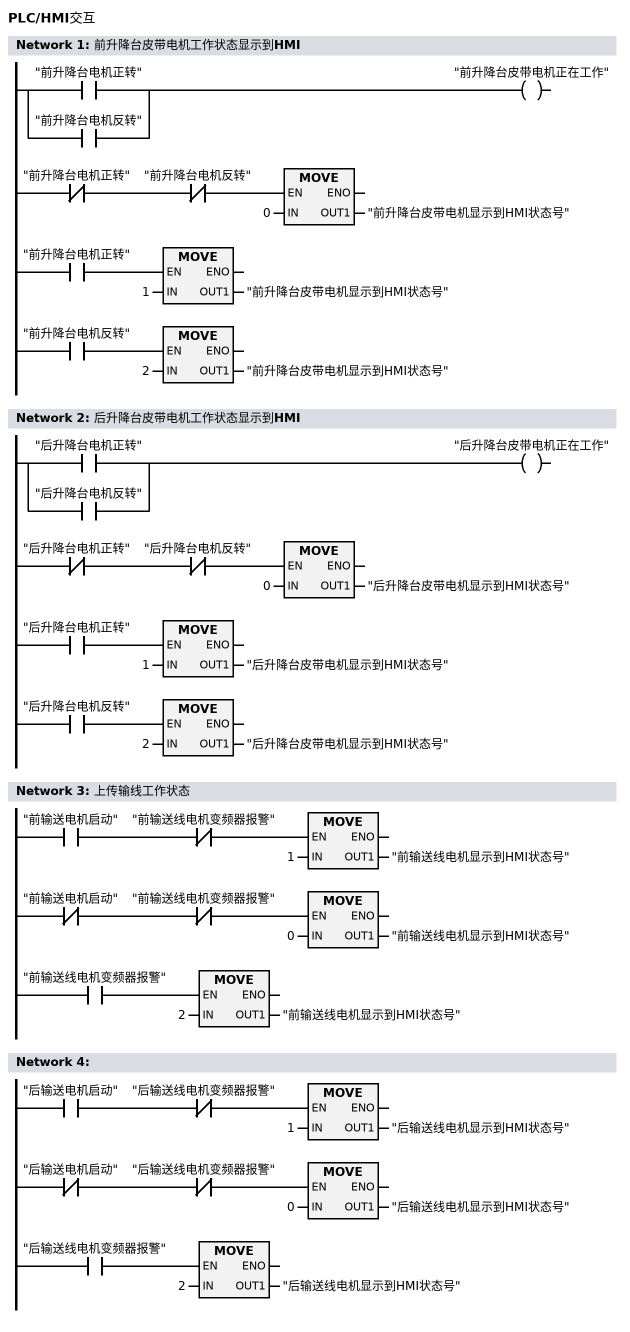
   RUNG wire#powerrail
      Contact( "前升降台电机正转" )
      wire#w1
      Coil( "前升降台皮带电机正在工作" )
   END_RUNG
   RUNG wire#powerrail
      Contact( "前升降台电机反转" )
   END_RUNG wire#w1
   RUNG wire#powerrail
      I_Contact( "前升降台电机正转" )
      I_Contact( "前升降台电机反转" )
      Move(in := 0, out1 => "前升降台皮带电机显示到HMI状态号")
   END_RUNG
   RUNG wire#powerrail
      Contact( "前升降台电机正转" )
      Move(in := 1, out1 => "前升降台皮带电机显示到HMI状态号")
   END_RUNG
   RUNG wire#powerrail
      Contact( "前升降台电机反转" )
      Move(in := 2, out1 => "前升降台皮带电机显示到HMI状态号")
   END_RUNG
   // the same network as SCL:
   "前升降台皮带电机正在工作" := "前升降台电机正转" OR "前升降台电机反转";
   IF NOT "前升降台电机正转" AND NOT "前升降台电机反转" THEN "前升降台皮带电机显示到HMI状态号" := 0; END_IF;
   IF "前升降台电机正转" THEN "前升降台皮带电机显示到HMI状态号" := 1; END_IF;
   IF "前升降台电机反转" THEN "前升降台皮带电机显示到HMI状态号" := 2; END_IF;
END_REGION

REGION Network 2: 后升降台皮带电机工作状态显示到HMI
   RUNG wire#powerrail
      Contact( "后升降台电机正转" )
      wire#w1
      Coil( "后升降台皮带电机正在工作" )
   END_RUNG
   RUNG wire#powerrail
      Contact( "后升降台电机反转" )
   END_RUNG wire#w1
   RUNG wire#powerrail
      I_Contact( "后升降台电机正转" )
      I_Contact( "后升降台电机反转" )
      Move(in := 0, out1 => "后升降台皮带电机显示到HMI状态号")
   END_RUNG
   RUNG wire#powerrail
      Contact( "后升降台电机正转" )
      Move(in := 1, out1 => "后升降台皮带电机显示到HMI状态号")
   END_RUNG
   RUNG wire#powerrail
      Contact( "后升降台电机反转" )
      Move(in := 2, out1 => "后升降台皮带电机显示到HMI状态号")
   END_RUNG
   // the same network as SCL:
   "后升降台皮带电机正在工作" := "后升降台电机正转" OR "后升降台电机反转";
   IF NOT "后升降台电机正转" AND NOT "后升降台电机反转" THEN "后升降台皮带电机显示到HMI状态号" := 0; END_IF;
   IF "后升降台电机正转" THEN "后升降台皮带电机显示到HMI状态号" := 1; END_IF;
   IF "后升降台电机反转" THEN "后升降台皮带电机显示到HMI状态号" := 2; END_IF;
END_REGION

REGION Network 3: 上传输线工作状态
   RUNG wire#powerrail
      Contact( "前输送电机启动" )
      I_Contact( "前输送线电机变频器报警" )
      Move(in := 1, out1 => "前输送线电机显示到HMI状态号")
   END_RUNG
   RUNG wire#powerrail
      I_Contact( "前输送电机启动" )
      I_Contact( "前输送线电机变频器报警" )
      Move(in := 0, out1 => "前输送线电机显示到HMI状态号")
   END_RUNG
   RUNG wire#powerrail
      Contact( "前输送线电机变频器报警" )
      Move(in := 2, out1 => "前输送线电机显示到HMI状态号")
   END_RUNG
   // the same network as SCL:
   IF "前输送电机启动" AND NOT "前输送线电机变频器报警" THEN "前输送线电机显示到HMI状态号" := 1; END_IF;
   IF NOT "前输送电机启动" AND NOT "前输送线电机变频器报警" THEN "前输送线电机显示到HMI状态号" := 0; END_IF;
   IF "前输送线电机变频器报警" THEN "前输送线电机显示到HMI状态号" := 2; END_IF;
END_REGION

REGION Network 4
   RUNG wire#powerrail
      Contact( "后输送电机启动" )
      I_Contact( "后输送线电机变频器报警" )
      Move(in := 1, out1 => "后输送线电机显示到HMI状态号")
   END_RUNG
   RUNG wire#powerrail
      I_Contact( "后输送电机启动" )
      I_Contact( "后输送线电机变频器报警" )
      Move(in := 0, out1 => "后输送线电机显示到HMI状态号")
   END_RUNG
   RUNG wire#powerrail
      Contact( "后输送线电机变频器报警" )
      Move(in := 2, out1 => "后输送线电机显示到HMI状态号")
   END_RUNG
   // the same network as SCL:
   IF "后输送电机启动" AND NOT "后输送线电机变频器报警" THEN "后输送线电机显示到HMI状态号" := 1; END_IF;
   IF NOT "后输送电机启动" AND NOT "后输送线电机变频器报警" THEN "后输送线电机显示到HMI状态号" := 0; END_IF;
   IF "后输送线电机变频器报警" THEN "后输送线电机显示到HMI状态号" := 2; END_IF;
END_REGION
END_FUNCTION

FUNCTION "报警程序" : Void   // FC5, LAD
{ S7_Optimized_Access := 'TRUE' }
VERSION : 0.1
BEGIN

REGION Network 1: 前升降台升降气缸动作超时报警
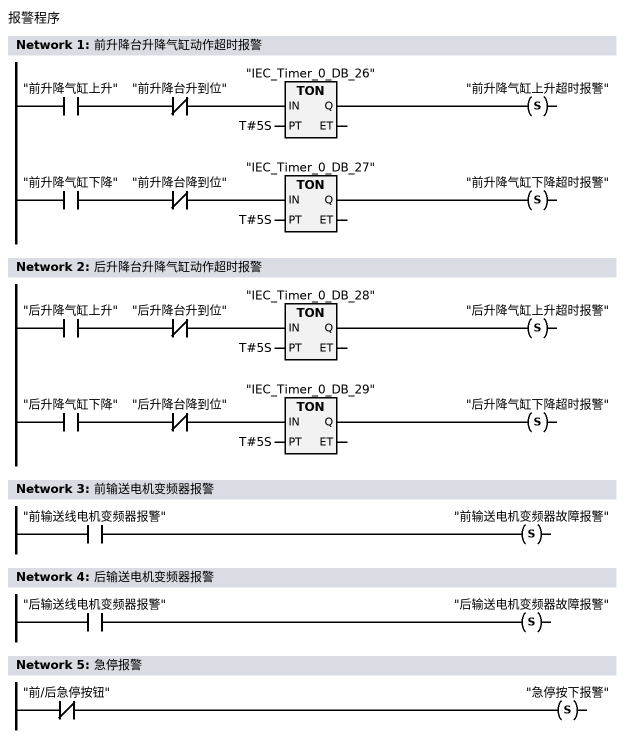
   "IEC_Timer_0_DB_26".TON(IN := "前升降气缸上升" AND NOT "前升降台升到位", PT := T#5S);
   IF "IEC_Timer_0_DB_26".Q THEN "前升降气缸上升超时报警" := TRUE; END_IF;
   "IEC_Timer_0_DB_27".TON(IN := "前升降气缸下降" AND NOT "前升降台降到位", PT := T#5S);
   IF "IEC_Timer_0_DB_27".Q THEN "前升降气缸下降超时报警" := TRUE; END_IF;
END_REGION

REGION Network 2: 后升降台升降气缸动作超时报警
   "IEC_Timer_0_DB_28".TON(IN := "后升降气缸上升" AND NOT "后升降台升到位", PT := T#5S);
   IF "IEC_Timer_0_DB_28".Q THEN "后升降气缸上升超时报警" := TRUE; END_IF;
   "IEC_Timer_0_DB_29".TON(IN := "后升降气缸下降" AND NOT "后升降台降到位", PT := T#5S);
   IF "IEC_Timer_0_DB_29".Q THEN "后升降气缸下降超时报警" := TRUE; END_IF;
END_REGION

REGION Network 3: 前输送电机变频器报警
   RUNG wire#powerrail
      Contact( "前输送线电机变频器报警" )
      S_Coil( "前输送电机变频器故障报警" )
   END_RUNG
   // the same network as SCL:
   IF "前输送线电机变频器报警" THEN "前输送电机变频器故障报警" := TRUE; END_IF;
END_REGION

REGION Network 4: 后输送电机变频器报警
   RUNG wire#powerrail
      Contact( "后输送线电机变频器报警" )
      S_Coil( "后输送电机变频器故障报警" )
   END_RUNG
   // the same network as SCL:
   IF "后输送线电机变频器报警" THEN "后输送电机变频器故障报警" := TRUE; END_IF;
END_REGION

REGION Network 5: 急停报警
   RUNG wire#powerrail
      I_Contact( "前/后急停按钮" )
      S_Coil( "急停按下报警" )
   END_RUNG
   // the same network as SCL:
   IF NOT "前/后急停按钮" THEN "急停按下报警" := TRUE; END_IF;
END_REGION
END_FUNCTION

FUNCTION "设备状态" : Void   // FC6, LAD
{ S7_Optimized_Access := 'TRUE' }
VERSION : 0.1
BEGIN

REGION Network 1: 急停拍下
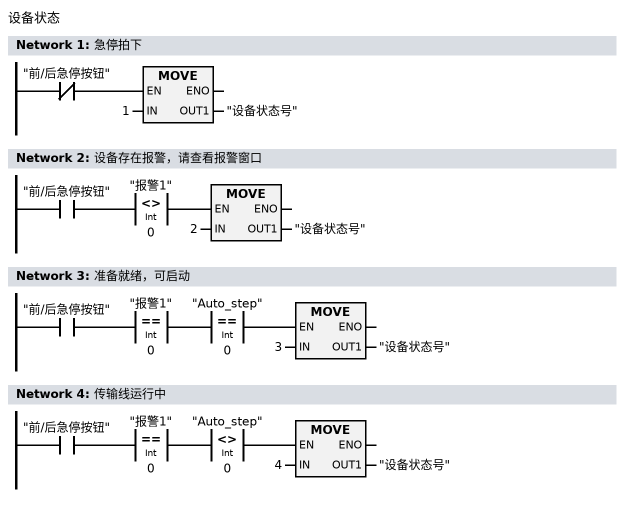
   RUNG wire#powerrail
      I_Contact( "前/后急停按钮" )
      Move(in := 1, out1 => "设备状态号")
   END_RUNG
   // the same network as SCL:
   IF NOT "前/后急停按钮" THEN "设备状态号" := 1; END_IF;
END_REGION

REGION Network 2: 设备存在报警，请查看报警窗口
   RUNG wire#powerrail
      Contact( "前/后急停按钮" )
      { S7_Templates := "SrcType := Int" } NE_Contact(in1 := "报警1", in2 := 0)
      Move(in := 2, out1 => "设备状态号")
   END_RUNG
   // the same network as SCL:
   IF "前/后急停按钮" AND ("报警1" <> 0) THEN "设备状态号" := 2; END_IF;
END_REGION

REGION Network 3: 准备就绪，可启动
   RUNG wire#powerrail
      Contact( "前/后急停按钮" )
      { S7_Templates := "SrcType := Int" } EQ_Contact(in1 := "报警1", in2 := 0)
      { S7_Templates := "SrcType := Int" } EQ_Contact(in1 := "Auto_step", in2 := 0)
      Move(in := 3, out1 => "设备状态号")
   END_RUNG
   // the same network as SCL:
   IF "前/后急停按钮" AND ("报警1" = 0) AND ("Auto_step" = 0) THEN "设备状态号" := 3; END_IF;
END_REGION

REGION Network 4: 传输线运行中
   RUNG wire#powerrail
      Contact( "前/后急停按钮" )
      { S7_Templates := "SrcType := Int" } EQ_Contact(in1 := "报警1", in2 := 0)
      { S7_Templates := "SrcType := Int" } NE_Contact(in1 := "Auto_step", in2 := 0)
      Move(in := 4, out1 => "设备状态号")
   END_RUNG
   // the same network as SCL:
   IF "前/后急停按钮" AND ("报警1" = 0) AND ("Auto_step" <> 0) THEN "设备状态号" := 4; END_IF;
END_REGION
END_FUNCTION

ORGANIZATION_BLOCK "Main"   // OB1, LAD, ProgramCycle
TITLE = "Main Program Sweep (Cycle)"
{ S7_Optimized_Access := 'TRUE' }
VERSION : 0.1
   VAR_INPUT
      Initial_Call : Bool;   // Initial call of this OB
      Remanence : Bool;   // =True, if remanent data are available
   END_VAR
   VAR_TEMP   // added for the SCL form of the ladder/FBD networks
      _w1 : Bool;
      _w2 : Bool;
      _w3 : Bool;
   END_VAR
BEGIN

REGION Network 1: MODBUS
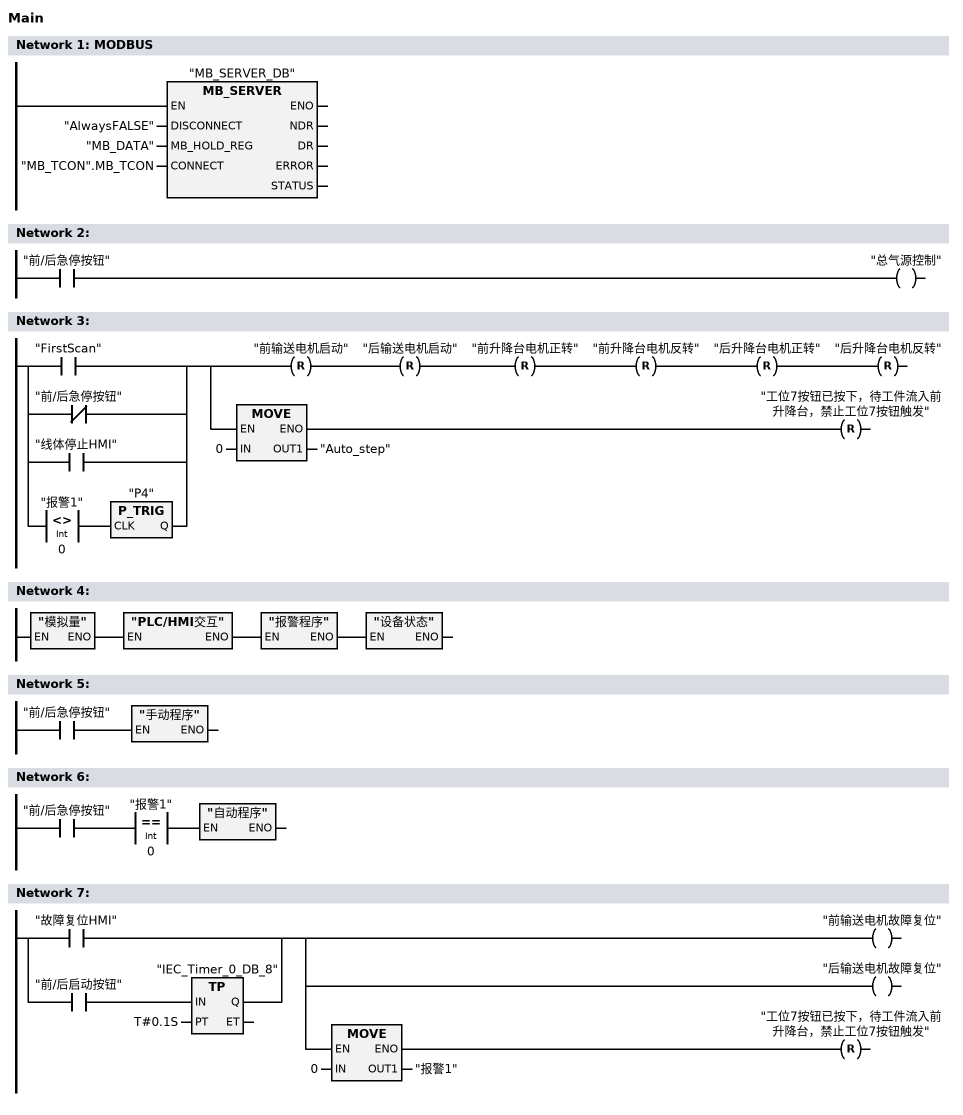
   "MB_SERVER_DB"(DISCONNECT := "AlwaysFALSE", MB_HOLD_REG := "MB_DATA", CONNECT := "MB_TCON".MB_TCON);   // MB_SERVER
END_REGION

REGION Network 2
   RUNG wire#powerrail
      Contact( "前/后急停按钮" )
      Coil( "总气源控制" )
   END_RUNG
   // the same network as SCL:
   "总气源控制" := "前/后急停按钮";
END_REGION

REGION Network 3
   RUNG wire#powerrail
      Contact( "FirstScan" )
      wire#w1
      R_Coil( "前输送电机启动" )
      R_Coil( "后输送电机启动" )
      R_Coil( "前升降台电机正转" )
      R_Coil( "前升降台电机反转" )
      R_Coil( "后升降台电机正转" )
      R_Coil( "后升降台电机反转" )
   END_RUNG
   RUNG wire#powerrail
      I_Contact( "前/后急停按钮" )
   END_RUNG wire#w1
   RUNG wire#powerrail
      Contact( "线体停止HMI" )
   END_RUNG wire#w1
   RUNG wire#powerrail
      { S7_Templates := "SrcType := Int" } NE_Contact(in1 := "报警1", in2 := 0)
      P_Trig( "P4" )
   END_RUNG wire#w1
   RUNG wire#w1
      Move(in := 0, out1 => "Auto_step")
      R_Coil( "工位7按钮已按下，待工件流入前升降台，禁止工位7按钮触发" )
   END_RUNG
   // the same network as SCL:
   #_w1 := "报警1" <> 0;
   #_w2 := #_w1 AND NOT "P4";   // rising edge
   "P4" := #_w1;
   IF "FirstScan" OR NOT "前/后急停按钮" OR "线体停止HMI" OR #_w2 THEN
       "前输送电机启动" := FALSE;
       "后输送电机启动" := FALSE;
       "前升降台电机正转" := FALSE;
       "前升降台电机反转" := FALSE;
       "后升降台电机正转" := FALSE;
       "后升降台电机反转" := FALSE;
       "Auto_step" := 0;
       "工位7按钮已按下，待工件流入前升降台，禁止工位7按钮触发" := FALSE;
   END_IF;
END_REGION

REGION Network 4
   RUNG wire#powerrail
      "模拟量"()
      "PLC/HMI交互"()
      "报警程序"()
      "设备状态"()
   END_RUNG
   // the same network as SCL:
   "模拟量"(ENO => #_w1);
   "PLC/HMI交互"(EN := #_w1, ENO => #_w2);
   "报警程序"(EN := #_w2, ENO => #_w3);
   IF #_w3 THEN "设备状态"(); END_IF;
END_REGION

REGION Network 5
   RUNG wire#powerrail
      Contact( "前/后急停按钮" )
      "手动程序"()
   END_RUNG
   // the same network as SCL:
   IF "前/后急停按钮" THEN "手动程序"(); END_IF;
END_REGION

REGION Network 6
   RUNG wire#powerrail
      Contact( "前/后急停按钮" )
      { S7_Templates := "SrcType := Int" } EQ_Contact(in1 := "报警1", in2 := 0)
      "自动程序"()
   END_RUNG
   // the same network as SCL:
   IF "前/后急停按钮" AND ("报警1" = 0) THEN "自动程序"(); END_IF;
END_REGION

REGION Network 7
   "IEC_Timer_0_DB_8".TP(IN := "前/后启动按钮", PT := T#0.1S);
   "前输送电机故障复位" := "故障复位HMI" OR "IEC_Timer_0_DB_8".Q;
   "后输送电机故障复位" := "前输送电机故障复位";
   IF "前输送电机故障复位" THEN
       "报警1" := 0;
       "工位7按钮已按下，待工件流入前升降台，禁止工位7按钮触发" := FALSE;
   END_IF;
END_REGION
END_ORGANIZATION_BLOCK

(* ===== HMI "HMI_RT_2" =====
system functions are stored by id; their names below are inferred from use
connection "HMI_连接_1": ETHERNET, SMART_S7_1200_OMS

HMI tags "默认变量表"
   "前/后急停按钮" : Bool = PLC "前/后急停按钮" AT %I0.0, 100 ms
   "前/后启动按钮" : Bool = PLC "前/后启动按钮" AT %I0.1, 100 ms
   "前输送线电机变频器报警" : Bool = PLC 前输送线电机变频器报警 AT %I0.2, 100 ms
   "后输送线电机变频器报警" : Bool = PLC 后输送线电机变频器报警 AT %I0.3, 100 ms
   "后方下轨道进料口有料检测" : Bool = PLC 后方下轨道进料口有料检测 AT %I0.4, 100 ms
   "后升降台有料检测" : Bool = PLC 后升降台有料检测 AT %I0.5, 100 ms
   "前方下轨道出料口有料检测" : Bool = PLC 前方下轨道出料口有料检测 AT %I0.6, 100 ms
   "前升降台有料检测" : Bool = PLC 前升降台有料检测 AT %I0.7, 100 ms
   "前升降台上轨道进料口料盘有料防呆检测" : Bool = PLC 备用2 AT %I1.0, 100 ms
   "前升降台升到位" : Bool = PLC 前升降台升到位 AT %I1.1, 100 ms
   "前升降台降到位" : Bool = PLC 前升降台降到位 AT %I1.2, 100 ms
   "后升降台升到位" : Bool = PLC 后升降台升到位 AT %I1.3, 100 ms
   "后升降台降到位" : Bool = PLC 后升降台降到位 AT %I1.4, 100 ms
   "备用1" : Bool = PLC 备用1 AT %I1.5, 100 ms
   "工位1放行按钮" : Bool = PLC 工位1放行按钮 AT %I2.0, 100 ms
   "工位2放行按钮" : Bool = PLC 工位2放行按钮 AT %I2.1, 100 ms
   "工位3放行按钮" : Bool = PLC 工位3放行按钮 AT %I2.2, 100 ms
   "工位4放行按钮" : Bool = PLC 工位4放行按钮 AT %I2.3, 100 ms
   "工位5放行按钮" : Bool = PLC 工位5放行按钮 AT %I2.4, 100 ms
   "工位6放行按钮" : Bool = PLC 工位6放行按钮 AT %I2.5, 100 ms
   "工位7放行按钮" : Bool = PLC 工位7放行按钮 AT %I2.6, 100 ms
   "备用2" : Bool = PLC 前升降台上轨道进料口料盘有料防呆检测 AT %I2.7, 100 ms
   "工位1光电检测" : Bool = PLC 工位1光电检测 AT %I3.0, 100 ms
   "工位2光电检测" : Bool = PLC 工位2光电检测 AT %I3.1, 100 ms
   "工位3光电检测" : Bool = PLC 工位3光电检测 AT %I3.2, 100 ms
   "工位4光电检测" : Bool = PLC 工位4光电检测 AT %I3.3, 100 ms
   "工位5光电检测" : Bool = PLC 工位5光电检测 AT %I3.4, 100 ms
   "工位6光电检测" : Bool = PLC 工位6光电检测 AT %I3.5, 100 ms
   "工位7光电检测" : Bool = PLC 工位7光电检测 AT %I3.6, 100 ms
   "备用3" : Bool = PLC 备用3 AT %I3.7, 100 ms
   "前输送电机启动" : Bool = PLC 前输送电机启动 AT %Q0.0, 100 ms
   "前输送电机故障复位" : Bool = PLC 前输送电机故障复位 AT %Q0.1, 100 ms
   "后输送电机启动" : Bool = PLC 后输送电机启动 AT %Q0.2, 100 ms
   "后输送电机故障复位" : Bool = PLC 后输送电机故障复位 AT %Q0.3, 100 ms
   "前升降台电机正转" : Bool = PLC 前升降台电机正转 AT %Q0.4, 100 ms
   "前升降台电机反转" : Bool = PLC 前升降台电机反转 AT %Q0.5, 100 ms
   "后升降台电机正转" : Bool = PLC 后升降台电机正转 AT %Q0.6, 100 ms
   "后升降台电机反转" : Bool = PLC 后升降台电机反转 AT %Q0.7, 100 ms
   "总气源控制" : Bool = PLC 总气源控制 AT %Q1.0, 100 ms
   "工位3阻挡气缸上升" : Bool = PLC 工位3阻挡气缸上升 AT %Q1.1, 100 ms
   "工位1阻挡气缸下降" : Bool = PLC 工位1阻挡气缸下降 AT %Q2.0, 100 ms
   "工位2阻挡气缸下降" : Bool = PLC 工位2阻挡气缸下降 AT %Q2.1, 100 ms
   "工位3阻挡气缸下降" : Bool = PLC 工位3阻挡气缸下降 AT %Q2.2, 100 ms
   "工位4阻挡气缸下降" : Bool = PLC 工位4阻挡气缸下降 AT %Q2.3, 100 ms
   "工位5阻挡气缸下降" : Bool = PLC 工位5阻挡气缸下降 AT %Q2.4, 100 ms
   "工位6阻挡气缸下降" : Bool = PLC 工位6阻挡气缸下降 AT %Q2.5, 100 ms
   "工位7阻挡气缸下降" : Bool = PLC 工位7阻挡气缸下降 AT %Q2.6, 100 ms
   "后方下轨道进料口阻挡气缸下降" : Bool = PLC 后方下轨道进料口阻挡气缸下降 AT %Q2.7, 100 ms
   "前升降气缸上升" : Bool = PLC 前升降气缸上升 AT %Q3.0, 100 ms
   "前升降气缸下降" : Bool = PLC 前升降气缸下降 AT %Q3.1, 100 ms
   "后升降气缸上升" : Bool = PLC 后升降气缸上升 AT %Q3.2, 100 ms
   "后升降气缸下降" : Bool = PLC 后升降气缸下降 AT %Q3.3, 100 ms
   "后方下轨道阻挡气缸上升" : Bool = PLC 后方下轨道阻挡气缸下降 AT %Q3.4, 100 ms
   "后方下轨道阻挡气缸下降" : Bool = PLC 后方下轨道阻挡气缸上升 AT %Q3.5, 100 ms
   "工位4阻挡气缸上升" : Bool = PLC 工位4阻挡气缸上升 AT %Q3.6, 100 ms
   "工位5阻挡气缸上升" : Bool = PLC 工位5阻挡气缸上升 AT %Q3.7, 100 ms
   "保持数据块_产品型号" : Int = PLC 保持数据块.产品型号 AT %DB23.DBW0, 100 ms
   "前输送线电机启动HMI" : Bool = PLC 前输送线电机启动HMI AT %M10.0, 100 ms
   "前输送线电机停止HMI" : Bool = PLC 前输送线电机停止HMI AT %M10.1, 100 ms
   "后输送线电机启动HMI" : Bool = PLC 后输送线电机启动HMI AT %M10.2, 100 ms
   "后输送线电机停止HMI" : Bool = PLC 后输送线电机停止HMI AT %M10.3, 100 ms
   "前升降台内部电机正转HMI" : Bool = PLC 前升降台内部电机正转HMI AT %M10.4, 100 ms
   "前升降台内部电机反转HMI" : Bool = PLC 前升降台内部电机反转HMI AT %M10.5, 100 ms
   "前升降台内部电机停止运行HMI" : Bool = PLC 前升降台内部电机停止运行HMI AT %M10.6, 100 ms
   "后升降台内部电机正转HMI" : Bool = PLC 后升降台内部电机正转HMI AT %M10.7, 100 ms
   "后升降台内部电机反转HMI" : Bool = PLC 后升降台内部电机反转HMI AT %M11.0, 100 ms
   "后升降台内部电机停止运行HMI" : Bool = PLC 后升降台内部电机停止运行HMI AT %M11.1, 100 ms
   "前升降气缸上升HMI" : Bool = PLC 前升降气缸上升HMI AT %M11.2, 100 ms
   "前升降气缸下降HMI" : Bool = PLC 前升降气缸下降HMI AT %M11.3, 100 ms
   "后升降气缸上升HMI" : Bool = PLC 后升降气缸上升HMI AT %M11.4, 100 ms
   "后升降气缸下降HMI" : Bool = PLC 后升降气缸下降HMI AT %M11.5, 100 ms
   "工位1阻挡气缸上升HMI" : Bool = PLC 工位1阻挡气缸上升HMI AT %M11.6, 100 ms
   "工位1阻挡气缸下降HMI" : Bool = PLC 工位1阻挡气缸下降HMI AT %M11.7, 100 ms
   "工位2阻挡气缸上升HMI" : Bool = PLC 工位2阻挡气缸上升HMI AT %M12.0, 100 ms
   "工位2阻挡气缸下降HMI" : Bool = PLC 工位2阻挡气缸下降HMI AT %M12.1, 100 ms
   "工位3阻挡气缸上升HMI" : Bool = PLC 工位3阻挡气缸上升HMI AT %M12.2, 100 ms
   "工位3阻挡气缸下降HMI" : Bool = PLC 工位3阻挡气缸下降HMI AT %M12.3, 100 ms
   "工位4阻挡气缸上升HMI" : Bool = PLC 工位4阻挡气缸上升HMI AT %M12.4, 100 ms
   "工位4阻挡气缸下降HMI" : Bool = PLC 工位4阻挡气缸下降HMI AT %M12.5, 100 ms
   "工位5阻挡气缸上升HMI" : Bool = PLC 工位5阻挡气缸上升HMI AT %M12.6, 100 ms
   "工位5阻挡气缸下降HMI" : Bool = PLC 工位5阻挡气缸下降HMI AT %M12.7, 100 ms
   "工位6阻挡气缸上升HMI" : Bool = PLC 工位6阻挡气缸上升HMI AT %M13.0, 100 ms
   "工位6阻挡气缸下降HMI" : Bool = PLC 工位6阻挡气缸下降HMI AT %M13.1, 100 ms
   "工位7阻挡气缸上升HMI" : Bool = PLC 工位7阻挡气缸上升HMI AT %M13.2, 100 ms
   "工位7阻挡气缸下降HMI" : Bool = PLC 工位7阻挡气缸下降HMI AT %M13.3, 100 ms
   "线体启动HMI" : Bool = PLC 线体启动HMI AT %M20.0, 100 ms
   "线体停止HMI" : Bool = PLC 线体停止HMI AT %M20.1, 100 ms
   "前升降台皮带电机正在工作" : Bool = PLC 前升降台皮带电机正在工作 AT %M100.0, 100 ms
   "后升降台皮带电机正在工作" : Bool = PLC 后升降台皮带电机正在工作 AT %M100.1, 100 ms
   "保持数据块_前输送电机变频器设定频率" : Int = PLC 保持数据块.前输送电机变频器设定频率 AT %DB23.DBW2, 100 ms
   "保持数据块_后输送电机变频器设定频率" : Int = PLC 保持数据块.后输送电机变频器设定频率 AT %DB23.DBW4, 100 ms
   "前升降台皮带电机显示到HMI状态号" : Word = PLC 前升降台皮带电机显示到HMI状态号 AT %MW2000, 100 ms
   "后升降台皮带电机显示到HMI状态号" : Int = PLC 后升降台皮带电机显示到HMI状态号 AT %MW2002, 100 ms
   "前输送线电机显示到HMI状态号" : Int = PLC 前输送线电机显示到HMI状态号 AT %MW2004, 100 ms
   "后输送线电机显示到HMI状态号" : Int = PLC 后输送线电机显示到HMI状态号 AT %MW2006, 100 ms
   "故障复位HMI" : Bool = PLC 故障复位HMI AT %M20.2, 100 ms
   "保持数据块_手动放行/自动放行" : Bool = PLC 保持数据块.手动放行/自动放行 AT %DB23.DBX6.0, 100 ms
   "报警1" : Int = PLC 报警1 AT %MW1000, 100 ms
   "设备状态号" : Int = PLC 设备状态号 AT %MW54, 100 ms
   "后方下轨道进料口阻挡气缸上升HMI" : Bool = PLC 后方下轨道进料口阻挡气缸上升HMI AT %M13.4, 100 ms
   "后方下轨道进料口阻挡气缸下降HMI" : Bool = PLC 后方下轨道进料口阻挡气缸下降HMI AT %M13.5, 100 ms
   "后方下轨道阻挡气缸上升HMI" : Bool = PLC 后方下轨道阻挡气缸上升HMI AT %M13.6, 100 ms
   "后方下轨道阻挡气缸下降HMI" : Bool = PLC 后方下轨道阻挡气缸下降HMI AT %M13.7, 100 ms
   "密码" : WString[254] AT %DB1.DBX0.0
   "用户名" : WString[254] AT %DB1.DBX0.0
   "编号" : Int AT %DB1.DBW0
   "滑移力检测工位" : Int = PLC 保持数据块.滑移力检测工位 AT %DB23.DBW8, 1 s
   "上柱管轴承压装工位" : Int = PLC 保持数据块.上柱管轴承压装工位 AT %DB23.DBW10, 1 s
   "拉轴工位" : Int = PLC 保持数据块.拉轴工位 AT %DB23.DBW12, 1 s
   "手柄装配工位" : Int = PLC 保持数据块.手柄装配工位 AT %DB23.DBW14, 1 s
   "上下柱管压装工位" : Int = PLC 保持数据块.上下柱管压装工位 AT %DB23.DBW16, 1 s
   "滑移力复测工位" : Int = PLC 保持数据块.滑移力复测工位 AT %DB23.DBW18, 1 s
   "调节机构检测工位" : Int = PLC 保持数据块.手柄调节机构工位 AT %DB23.DBW20, 1 s

discrete alarms
   1: '前升降气缸上升超时报警！！！', class Errors, trigger "报警1" bit 8
   2: '前升降气缸下降超时报警！！！', class Errors, trigger "报警1" bit 9
   3: '后升降气缸上升超时报警！！！', class Errors, trigger "报警1" bit 10
   4: '后升降气缸下降超时报警！！！', class Errors, trigger "报警1" bit 11
   5: '上输送线电机故障报警！！！', class Errors, trigger "报警1" bit 12
   6: '下输送线电机故障报警！！！', class Errors, trigger "报警1" bit 13
   7: '急停拍下报警！！！', class Errors, trigger "报警1" bit 14

text list "产品型号": 1 'R92A'; 2 'R128'; 3 'R527'; 4 'R538'; 5 'R563X'; 6 'R567X'; 7 '备用2'; 8 '备用3'; 9 '备用4'; 10 '备用5'

text list "前升降皮带工作状态": 0 '停止'; 1 '正转'; 2 '反转'

text list "后升降皮带工作状态": 0 '停止'; 1 '正转'; 2 '反转'

text list "设备状态显示": 1 '急停拍下！！！'; 2 '设备存在报警，请查看报警窗口！！！'; 3 '准备就绪，可启动'; 4 '传输线运行中'

text list "上输送线工作状态": 0 '上传输线停止'; 1 '上传输线运行'; 2 '上传输线报警'

text list "下输送线工作状态": 0 '下传输线停止'; 1 '下传输线运行'; 2 '下传输线报警'

recipe "传输线参数写入": 滑移力检测工位 <- "滑移力检测工位", 上柱管轴承压装工位 <- "上柱管轴承压装工位", 拉轴工位 <- "拉轴工位", 手柄装配工位 <- "手柄装配工位", 上下柱管压装工位 <- "上下柱管压装工位", 滑移力复测工位 <- "滑移力复测工位", Recipe_element_1 <- "调节机构检测工位"

screen "DI_1" 800x480, template "模板"
   TextField "文本域_1" at 0,0 size 800x50; Text 'DI_1'
   Button "在线_2" at 16,82 size 85x39; TextOn 'DI监控1'; TextOff 'DI监控1'
      on Release: ActivateScreen("DI_1", 0)
   Button "在线_3" at 16,133 size 85x39; TextOn 'DI监控2'; TextOff 'DI监控2'
      on Release: ActivateScreen("DI_2", 0)
   Circle "圆_3" at 179,80 size 24x24
      Appearance <- "前/后急停按钮"
   TextField "文本域_12" at 217,79 size 144x26; Text 'I0.0 前/后急停按钮'
   TextField "文本域_3" at 217,123 size 144x26; Text 'I0.1 前/后启动按钮'
   TextField "文本域_4" at 217,167 size 216x26; Text 'I0.2 前输送线电机变频器报警'
   TextField "文本域_5" at 217,212 size 216x26; Text 'I0.3 后输送线电机变频器报警'
   TextField "文本域_6" at 217,256 size 200x26; Text 'I0.4 下轨道进料口有料检测'
   TextField "文本域_7" at 217,301 size 168x26; Text 'I0.5 前升降台有料检测'
   TextField "文本域_8" at 217,345 size 168x26; Text 'I0.6 后升降台有料检测'
   TextField "文本域_9" at 217,390 size 200x26; Text 'I0.7 下轨道出料口有料检测'
   Circle "圆_2" at 179,124 size 24x24
      Appearance <- "前/后启动按钮"
   TextField "文本域_10" at 529,79 size 72x26; Text 'I1.0 备用'
   TextField "文本域_11" at 529,123 size 152x26; Text 'I1.1 前升降台升到位'
   TextField "文本域_13" at 529,167 size 152x26; Text 'I1.2 前升降台降到位'
   TextField "文本域_14" at 529,212 size 152x26; Text 'I1.3 后升降台升到位'
   TextField "文本域_15" at 529,256 size 152x26; Text 'I1.4 后升降台降到位'
   TextField "文本域_16" at 529,301 size 72x26; Text 'I1.5 备用'
   Circle "圆_4" at 179,168 size 24x24
      Appearance <- "前输送线电机变频器报警"
   Circle "圆_5" at 179,213 size 24x24
      Appearance <- "后输送线电机变频器报警"
   Circle "圆_6" at 179,257 size 24x24
      Appearance <- "后方下轨道进料口有料检测"
   Circle "圆_7" at 179,302 size 24x24
      Appearance <- "前升降台有料检测"
   Circle "圆_8" at 179,346 size 24x24
      Appearance <- "后升降台有料检测"
   Circle "圆_9" at 179,391 size 24x24
      Appearance <- "前方下轨道出料口有料检测"
   Circle "圆_10" at 493,80 size 24x24
      Appearance <- "前升降台上轨道进料口料盘有料防呆检测"
   Circle "圆_11" at 493,124 size 24x24
      Appearance <- "前升降台升到位"
   Circle "圆_12" at 493,168 size 24x24
      Appearance <- "前升降台降到位"
   Circle "圆_13" at 493,213 size 24x24
      Appearance <- "后升降台升到位"
   Circle "圆_14" at 493,257 size 24x24
      Appearance <- "后升降台降到位"
   Circle "圆_15" at 493,302 size 24x24
      Appearance <- "备用1"
   Button "在线_1" at 16,272 size 85x39; TextOn 'DO监控1'; TextOff 'DO监控1'
      on Release: ActivateScreen("DO_1", 0)
   Button "在线_5" at 16,323 size 85x39; TextOn 'DO监控2'; TextOff 'DO监控2'
      on Release: ActivateScreen("DO_2", 0)

screen "DI_2" 800x480, template "模板"
   TextField "文本域_17" at 217,81 size 146x26; Text 'I2.0 工位1放行按钮'
   TextField "文本域_18" at 217,125 size 146x26; Text 'I2.1 工位2放行按钮'
   TextField "文本域_19" at 217,169 size 146x26; Text 'I2.2 工位3放行按钮'
   TextField "文本域_20" at 217,214 size 146x26; Text 'I2.3 工位4放行按钮'
   TextField "文本域_21" at 217,258 size 146x26; Text 'I2.4 工位5放行按钮'
   TextField "文本域_22" at 217,303 size 146x26; Text 'I2.5 工位6放行按钮'
   TextField "文本域_23" at 217,347 size 146x26; Text 'I2.6 工位7放行按钮'
   TextField "文本域_24" at 217,392 size 232x26; Text 'I2.7 前升降台料盘有料防呆检测'
   Circle "圆_17" at 179,81 size 24x24
      Appearance <- "工位1放行按钮"
   Circle "圆_18" at 179,125 size 24x24
      Appearance <- "工位2放行按钮"
   Circle "圆_19" at 179,169 size 24x24
      Appearance <- "工位3放行按钮"
   Circle "圆_20" at 179,214 size 24x24
      Appearance <- "工位4放行按钮"
   Circle "圆_21" at 179,258 size 24x24
      Appearance <- "工位5放行按钮"
   Circle "圆_22" at 179,303 size 24x24
      Appearance <- "工位6放行按钮"
   Circle "圆_23" at 179,347 size 24x24
      Appearance <- "工位7放行按钮"
   Circle "圆_24" at 179,392 size 24x24
      Appearance <- "备用2"
   Circle "圆_2" at 493,81 size 24x24
      Appearance <- "工位1光电检测"
   TextField "文本域_3" at 529,81 size 146x26; Text 'I3.0 工位1光电检测'
   TextField "文本域_4" at 529,125 size 146x26; Text 'I3.1 工位2光电检测'
   TextField "文本域_5" at 529,169 size 146x26; Text 'I3.2 工位3光电检测'
   TextField "文本域_6" at 529,214 size 146x26; Text 'I3.3 工位4光电检测'
   TextField "文本域_7" at 529,258 size 146x26; Text 'I3.4 工位5光电检测'
   TextField "文本域_8" at 529,303 size 146x26; Text 'I3.5 工位6光电检测'
   TextField "文本域_9" at 529,347 size 146x26; Text 'I3.6 工位7光电检测'
   TextField "文本域_10" at 529,392 size 72x26; Text 'I3.7 备用'
   Circle "圆_3" at 493,125 size 24x24
      Appearance <- "工位2光电检测"
   Circle "圆_4" at 493,169 size 24x24
      Appearance <- "工位3光电检测"
   Circle "圆_5" at 493,214 size 24x24
      Appearance <- "工位4光电检测"
   Circle "圆_6" at 493,258 size 24x24
      Appearance <- "工位5光电检测"
   Circle "圆_7" at 493,303 size 24x24
      Appearance <- "工位6光电检测"
   Circle "圆_8" at 493,347 size 24x24
      Appearance <- "工位7光电检测"
   Circle "圆_9" at 493,392 size 24x24
      Appearance <- "备用3"
   TextField "文本域_1" at 0,0 size 800x50; Text 'DI_2'
   Button "在线_2" at 16,82 size 85x39; TextOn 'DI监控1'; TextOff 'DI监控1'
      on Release: ActivateScreen("DI_1", 0)
   Button "在线_3" at 16,133 size 85x39; TextOn 'DI监控2'; TextOff 'DI监控2'
      on Release: ActivateScreen("DI_2", 0)
   Button "在线_1" at 16,272 size 85x39; TextOn 'DO监控1'; TextOff 'DO监控1'
      on Release: ActivateScreen("DO_1", 0)
   Button "在线_5" at 16,323 size 85x39; TextOn 'DO监控2'; TextOff 'DO监控2'
      on Release: ActivateScreen("DO_2", 0)

screen "DO_1" 800x480, template "模板"
   Circle "圆_3" at 179,82 size 24x24
      Appearance <- "前输送电机启动"
   TextField "文本域_12" at 217,83 size 160x26; Text 'Q0.0 前输送电机启动'
   TextField "文本域_1" at 217,127 size 240x26; Text 'Q0.1 前输送电机变频器故障复位'
   TextField "文本域_3" at 217,171 size 160x26; Text 'Q0.2 后输送电机启动'
   TextField "文本域_4" at 217,215 size 240x26; Text 'Q0.3 后输送电机变频器故障复位'
   TextField "文本域_5" at 217,259 size 176x26; Text 'Q0.4 前升降台皮带正转'
   TextField "文本域_6" at 217,303 size 176x26; Text 'Q0.5 前升降台皮带反转'
   TextField "文本域_7" at 217,347 size 176x26; Text 'Q0.6 后升降台皮带正转'
   TextField "文本域_8" at 217,391 size 176x26; Text 'Q0.7 后升降台皮带反转'
   Circle "圆_2" at 179,126 size 24x24
      Appearance <- "前输送电机故障复位"
   TextField "文本域_9" at 531,83 size 128x26; Text 'Q1.0 总气源控制'
   TextField "文本域_10" at 531,127 size 186x26; Text 'Q1.1 工位3阻挡气缸上升'
   Circle "圆_4" at 179,170 size 24x24
      Appearance <- "后输送电机启动"
   Circle "圆_5" at 179,215 size 24x24
      Appearance <- "后输送电机故障复位"
   Circle "圆_6" at 179,259 size 24x24
      Appearance <- "前升降台电机正转"
   Circle "圆_7" at 179,304 size 24x24
      Appearance <- "前升降台电机反转"
   Circle "圆_8" at 179,348 size 24x24
      Appearance <- "后升降台电机正转"
   Circle "圆_9" at 179,393 size 24x24
      Appearance <- "后升降台电机反转"
   Circle "圆_10" at 493,82 size 24x24
      Appearance <- "总气源控制"
   Circle "圆_11" at 493,126 size 24x24
      Appearance <- "工位3阻挡气缸上升"
   TextField "文本域_2" at 0,0 size 800x50; Text 'DO_1'
   Button "在线_2" at 16,82 size 85x39; TextOn 'DI监控1'; TextOff 'DI监控1'
      on Release: ActivateScreen("DI_1", 0)
   Button "在线_3" at 16,133 size 85x39; TextOn 'DI监控2'; TextOff 'DI监控2'
      on Release: ActivateScreen("DI_2", 0)
   Button "在线_1" at 16,272 size 85x39; TextOn 'DO监控1'; TextOff 'DO监控1'
      on Release: ActivateScreen("DO_1", 0)
   Button "在线_5" at 16,323 size 85x39; TextOn 'DO监控2'; TextOff 'DO监控2'
      on Release: ActivateScreen("DO_2", 0)

screen "DO_2" 800x480, template "模板"
   TextField "文本域_17" at 217,81 size 186x26; Text 'Q2.0 工位1阻挡气缸下降'
   TextField "文本域_18" at 217,125 size 186x26; Text 'Q2.1 工位2阻挡气缸下降'
   TextField "文本域_19" at 217,170 size 186x26; Text 'Q2.2 工位3阻挡气缸下降'
   TextField "文本域_20" at 217,214 size 186x26; Text 'Q2.3 工位4阻挡气缸下降'
   TextField "文本域_21" at 217,259 size 186x26; Text 'Q2.4 工位5阻挡气缸下降'
   TextField "文本域_22" at 217,303 size 186x26; Text 'Q2.5 工位6阻挡气缸下降'
   TextField "文本域_23" at 217,348 size 186x26; Text 'Q2.6 工位7阻挡气缸下降'
   TextField "文本域_24" at 217,393 size 208x26; Text 'Q2.7 下进料口阻挡气缸下降'
   Circle "圆_17" at 179,82 size 24x24
      Appearance <- "工位1阻挡气缸下降"
   Circle "圆_18" at 179,126 size 24x24
      Appearance <- "工位2阻挡气缸下降"
   Circle "圆_2" at 179,170 size 24x24
      Appearance <- "工位3阻挡气缸下降"
   Circle "圆_3" at 179,215 size 24x24
      Appearance <- "工位4阻挡气缸下降"
   Circle "圆_21" at 179,259 size 24x24
      Appearance <- "工位5阻挡气缸下降"
   Circle "圆_22" at 179,304 size 24x24
      Appearance <- "工位6阻挡气缸下降"
   Circle "圆_23" at 179,348 size 24x24
      Appearance <- "工位7阻挡气缸下降"
   Circle "圆_24" at 179,393 size 24x24
      Appearance <- "后方下轨道进料口阻挡气缸下降"
   Circle "圆_4" at 493,82 size 24x24
      Appearance <- "前升降气缸上升"
   TextField "文本域_12" at 531,82 size 160x26; Text 'Q3.0 前升降气缸上升'
   TextField "文本域_1" at 531,126 size 160x26; Text 'Q3.1 前升降气缸下降'
   TextField "文本域_3" at 531,170 size 160x26; Text 'Q3.2 后升降气缸上升'
   TextField "文本域_4" at 531,214 size 160x26; Text 'Q3.3 后升降气缸下降'
   TextField "文本域_5" at 531,259 size 160x26; Text 'Q3.4 下阻挡气缸下降'
   TextField "文本域_6" at 531,303 size 160x26; Text 'Q3.5 下阻挡气缸上升'
   TextField "文本域_7" at 531,347 size 186x26; Text 'Q3.6 工位4阻挡气缸上升'
   TextField "文本域_8" at 531,392 size 186x26; Text 'Q3.7 工位5阻挡气缸上升'
   Circle "圆_5" at 493,126 size 24x24
      Appearance <- "前升降气缸下降"
   Circle "圆_6" at 493,170 size 24x24
      Appearance <- "后升降气缸上升"
   Circle "圆_7" at 493,215 size 24x24
      Appearance <- "后升降气缸下降"
   Circle "圆_8" at 493,259 size 24x24
      Appearance <- "后方下轨道阻挡气缸下降"
   Circle "圆_9" at 493,304 size 24x24
      Appearance <- "后方下轨道阻挡气缸上升"
   Circle "圆_10" at 493,348 size 24x24
      Appearance <- "工位4阻挡气缸上升"
   Circle "圆_11" at 493,393 size 24x24
      Appearance <- "工位5阻挡气缸上升"
   TextField "文本域_2" at 0,0 size 800x50; Text 'DO_2'
   Button "在线_2" at 16,82 size 85x39; TextOn 'DI监控1'; TextOff 'DI监控1'
      on Release: ActivateScreen("DI_1", 0)
   Button "在线_3" at 16,133 size 85x39; TextOn 'DI监控2'; TextOff 'DI监控2'
      on Release: ActivateScreen("DI_2", 0)
   Button "在线_1" at 16,272 size 85x39; TextOn 'DO监控1'; TextOff 'DO监控1'
      on Release: ActivateScreen("DO_1", 0)
   Button "在线_5" at 16,323 size 85x39; TextOn 'DO监控2'; TextOff 'DO监控2'
      on Release: ActivateScreen("DO_2", 0)

screen "登陆" 800x480, template "登陆"
   TextField "文本域_1" at 0,0 size 800x50; Text '传输线'

screen "输送线气缸" 800x480, template "模板"
   Button "在线_3" at 183,80 size 68x31; TextOn '放行'; TextOff '上升'
      on Release: ResetBit("工位1阻挡气缸上升HMI")
      on Press: SetBit("工位1阻挡气缸上升HMI")
   TextField "文本域_2" at 109,95 size 73x36; Text '工位1 阻挡气缸'
   Button "在线_6" at 183,114 size 68x31; TextOn '顶升'; TextOff '下降'
      on Release: ResetBit("工位1阻挡气缸下降HMI")
      on Press: SetBit("工位1阻挡气缸下降HMI")
   TextField "文本域_3" at 274,95 size 73x36; Text '工位2 阻挡气缸'
   TextField "文本域_4" at 439,97 size 73x36; Text '工位3 阻挡气缸'
   TextField "文本域_5" at 604,97 size 73x36; Text '工位4 阻挡气缸'
   Button "在线_7" at 349,80 size 68x31; TextOn '放行'; TextOff '上升'
      on Release: ResetBit("工位2阻挡气缸上升HMI")
      on Press: SetBit("工位2阻挡气缸上升HMI")
   Button "在线_8" at 349,114 size 68x31; TextOn '顶升'; TextOff '下降'
      on Release: ResetBit("工位2阻挡气缸下降HMI")
      on Press: SetBit("工位2阻挡气缸下降HMI")
   Button "在线_9" at 514,80 size 68x31; TextOn '放行'; TextOff '上升'
      on Release: ResetBit("工位3阻挡气缸上升HMI")
      on Press: SetBit("工位3阻挡气缸上升HMI")
   Button "在线_10" at 514,114 size 68x31; TextOn '顶升'; TextOff '下降'
      on Release: ResetBit("工位3阻挡气缸下降HMI")
      on Press: SetBit("工位3阻挡气缸下降HMI")
   Button "在线_11" at 678,80 size 68x31; TextOn '放行'; TextOff '上升'
      on Release: ResetBit("工位4阻挡气缸上升HMI")
      on Press: SetBit("工位4阻挡气缸上升HMI")
   Button "在线_12" at 678,114 size 68x31; TextOn '顶升'; TextOff '下降'
      on Release: ResetBit("工位4阻挡气缸下降HMI")
      on Press: SetBit("工位4阻挡气缸下降HMI")
   Button "在线_13" at 183,170 size 68x31; TextOn '放行'; TextOff '上升'
      on Release: ResetBit("工位5阻挡气缸上升HMI")
      on Press: SetBit("工位5阻挡气缸上升HMI")
   TextField "文本域_6" at 109,185 size 73x36; Text '工位5 阻挡气缸'
   Button "在线_14" at 183,204 size 68x31; TextOn '顶升'; TextOff '下降'
      on Release: ResetBit("工位5阻挡气缸下降HMI")
      on Press: SetBit("工位5阻挡气缸下降HMI")
   TextField "文本域_8" at 274,185 size 73x36; Text '工位6 阻挡气缸'
   TextField "文本域_10" at 439,187 size 73x36; Text '工位7 阻挡气缸'
   TextField "文本域_11" at 258,272 size 90x36; Text '下轨道进料 口阻挡气缸'
   Button "在线_15" at 349,170 size 68x31; TextOn '放行'; TextOff '上升'
      on Release: ResetBit("工位6阻挡气缸上升HMI")
      on Press: SetBit("工位6阻挡气缸上升HMI")
   Button "在线_16" at 349,204 size 68x31; TextOn '顶升'; TextOff '下降'
      on Release: ResetBit("工位6阻挡气缸下降HMI")
      on Press: SetBit("工位6阻挡气缸下降HMI")
   Button "在线_17" at 514,170 size 68x31; TextOn '放行'; TextOff '上升'
      on Release: ResetBit("工位7阻挡气缸上升HMI")
      on Press: SetBit("工位7阻挡气缸上升HMI")
   Button "在线_18" at 514,204 size 68x31; TextOn '顶升'; TextOff '下降'
      on Release: ResetBit("工位7阻挡气缸下降HMI")
      on Press: SetBit("工位7阻挡气缸下降HMI")
   Button "在线_19" at 350,255 size 68x31; TextOn '放行'; TextOff '上升'
      on Release: ResetBit("后方下轨道进料口阻挡气缸上升HMI")
      on Press: SetBit("后方下轨道进料口阻挡气缸上升HMI")
   Button "在线_20" at 350,289 size 68x31; TextOn '顶升'; TextOff '下降'
      on Release: ResetBit("后方下轨道进料口阻挡气缸下降HMI")
      on Press: SetBit("后方下轨道进料口阻挡气缸下降HMI")
   TextField "文本域_13" at 109,273 size 73x36; Text '下轨道 阻挡气缸'
   Button "在线_23" at 183,256 size 68x31; TextOn '放行'; TextOff '上升'
      on Release: ResetBit("后方下轨道阻挡气缸上升HMI")
      on Press: SetBit("后方下轨道阻挡气缸上升HMI")
   Button "在线_24" at 183,290 size 68x31; TextOn '顶升'; TextOff '下降'
      on Release: ResetBit("后方下轨道阻挡气缸下降HMI")
      on Press: SetBit("后方下轨道阻挡气缸下降HMI")
   Button "在线_21" at 271,333 size 68x31; TextOn '上升'; TextOff '上升'
      on Release: ResetBit("前升降气缸上升HMI")
      on Press: SetBit("前升降气缸上升HMI")
   TextField "文本域_12" at 197,332 size 73x36; Text '前升降 气缸上升'
   TextField "文本域_14" at 198,377 size 73x36; Text '前升降 气缸下降'
   TextField "文本域_15" at 503,332 size 73x36; Text '后升降 气缸上升'
   TextField "文本域_16" at 503,380 size 73x36; Text '后升降 气缸下降'
   Button "在线_25" at 271,381 size 68x31; TextOn '放行'; TextOff '下降'
      on Release: ResetBit("前升降气缸下降HMI")
      on Press: SetBit("前升降气缸下降HMI")
   Button "在线_27" at 576,335 size 68x31; TextOn '放行'; TextOff '上升'
      on Release: ResetBit("后升降气缸上升HMI")
      on Press: SetBit("后升降气缸上升HMI")
   Button "在线_29" at 576,381 size 68x31; TextOn '放行'; TextOff '下降'
      on Release: ResetBit("后升降气缸下降HMI")
      on Press: SetBit("后升降气缸下降HMI")
   Circle "圆_3" at 352,333 size 32x32
      Appearance <- "前升降台升到位"
   Circle "圆_2" at 352,381 size 32x32
      Appearance <- "前升降台降到位"
   Circle "圆_5" at 657,335 size 32x32
      Appearance <- "后升降台升到位"
   Circle "圆_7" at 657,381 size 32x32
      Appearance <- "后升降台降到位"
   TextField "文本域_9" at 0,0 size 800x50; Text '气缸手动操作'
   Button "在线_5" at 16,193 size 85x39; TextOn '输送线电机'; TextOff '输送线电机'
      on Release: ActivateScreen("输送线电机", 0)
   Button "在线_1" at 16,108 size 85x39; TextOn '输送线气缸'; TextOff '输送线气缸'
      on Release: ActivateScreen("输送线气缸", 0)

screen "输送线电机" 800x480, template "模板"
   Button "在线_5" at 16,193 size 85x39; TextOn '输送线电机'; TextOff '输送线电机'
      on Release: ActivateScreen("输送线电机", 0)
   Button "在线_7" at 16,108 size 85x39; TextOn '输送线气缸'; TextOff '输送线气缸'
      on Release: ActivateScreen("输送线气缸", 0)
   Button "在线_3" at 211,102 size 100x40; TextOn '启动'; TextOff '启动'
      on Release: ResetBit("前输送线电机启动HMI")
      on Press: SetBit("前输送线电机启动HMI")
   TextField "文本域_2" at 197,74 size 124x20; Text '前输送电机启动'
   Button "在线_6" at 211,197 size 100x40; TextOn '停止'; TextOff '停止'
      on Release: ResetBit("前输送线电机停止HMI")
      on Press: SetBit("前输送线电机停止HMI")
   TextField "文本域_3" at 197,169 size 124x20; Text '前输送电机停止'
   Button "在线_8" at 549,102 size 100x40; TextOn '启动'; TextOff '启动'
      on Release: ResetBit("后输送线电机启动HMI")
      on Press: SetBit("后输送线电机启动HMI")
   TextField "文本域_4" at 535,74 size 124x20; Text '后输送电机启动'
   Button "在线_9" at 549,197 size 100x40; TextOn '停止'; TextOff '停止'
      on Release: ResetBit("后输送线电机停止HMI")
      on Press: SetBit("后输送线电机停止HMI")
   TextField "文本域_5" at 535,169 size 124x20; Text '后输送电机停止'
   Button "在线_10" at 139,297 size 100x40; TextOn '正转'; TextOff '正转'
      on Release: ResetBit("前升降台内部电机正转HMI")
      on Press: SetBit("前升降台内部电机正转HMI")
   TextField "文本域_6" at 115,269 size 141x20; Text '前升降台皮带正转'
   Button "在线_11" at 211,384 size 100x40; TextOn '停止'; TextOff '停止'
      on Release: ResetBit("前升降台内部电机停止运行HMI")
      on Press: SetBit("前升降台内部电机停止运行HMI")
   TextField "文本域_8" at 192,356 size 141x20; Text '前输送线皮带停止'
   Button "在线_12" at 292,297 size 100x40; TextOn '反转'; TextOff '反转'
      on Release: ResetBit("前升降台内部电机反转HMI")
      on Press: SetBit("前升降台内部电机反转HMI")
   TextField "文本域_9" at 272,269 size 141x20; Text '前输送线皮带反转'
   Button "在线_13" at 466,297 size 100x40; TextOn '正转'; TextOff '正转'
      on Release: ResetBit("后升降台内部电机正转HMI")
      on Press: SetBit("后升降台内部电机正转HMI")
   TextField "文本域_10" at 445,269 size 141x20; Text '后输送线皮带正转'
   Button "在线_14" at 549,384 size 100x40; TextOn '停止'; TextOff '停止'
      on Release: ResetBit("后升降台内部电机停止运行HMI")
      on Press: SetBit("后升降台内部电机停止运行HMI")
   TextField "文本域_11" at 529,356 size 141x20; Text '后输送线皮带停止'
   Button "在线_15" at 625,297 size 100x40; TextOn '反转'; TextOff '反转'
      on Release: ResetBit("后升降台内部电机反转HMI")
      on Press: SetBit("后升降台内部电机反转HMI")
   TextField "文本域_12" at 603,269 size 141x20; Text '后输送线皮带反转'
   TextField "文本域_13" at 0,0 size 800x50; Text '电机手动操作'

screen "产品选择" 800x480, template "模板"
   TextField "文本域_4" at 0,0 size 800x50; Text '产品选择'
   SymbolicIOField "符号 I/O 域_1" at 182,86 size 111x46; TextOn '1'; TextOff '0'; TextList "产品型号"
      ProcessValue <- "保持数据块_产品型号"
   Button "在线_1" at 73,154 size 100x40; TextOn 'R92A'; TextOff 'R92A'
      on Press: function_eba64363(1, U 1, 1, N); function_b431313b(1, U 1, N); ActivateScreen("欢迎-管理员", 0); SetTag("保持数据块_产品型号", 1)
   Button "在线_2" at 207,154 size 100x40; TextOn 'R128'; TextOff 'R128'
      on Press: function_eba64363(1, U 2, 1, N); function_b431313b(1, U 2, N); ActivateScreen("欢迎-管理员", 0); SetTag("保持数据块_产品型号", 2)
   Button "在线_3" at 347,154 size 100x40; TextOn 'R527'; TextOff 'R527'
      on Press: function_eba64363(1, U 3, 1, N); function_b431313b(1, U 3, N); ActivateScreen("欢迎-管理员", 0); SetTag("保持数据块_产品型号", 3)
   Button "在线_4" at 488,154 size 100x40; TextOn 'R538'; TextOff 'R538'
      on Press: function_eba64363(1, U 4, 1, N); function_b431313b(1, U 4, N); ActivateScreen("欢迎-管理员", 0); SetTag("保持数据块_产品型号", 4)
   Button "在线_5" at 626,154 size 100x40; TextOn 'R544'; TextOff 'R563X'
      on Press: function_eba64363(1, U 5, 1, N); function_b431313b(1, U 5, N); ActivateScreen("欢迎-管理员", 0); SetTag("保持数据块_产品型号", 5)
   Button "在线_7" at 207,221 size 100x40; TextOn '在线'; TextOff '备用'
      on Release: SetTag("保持数据块_产品型号", 7); ActivateScreen("欢迎-管理员", 0)
   Button "在线_8" at 347,221 size 100x40; TextOn '在线'; TextOff '备用'
      on Release: SetTag("保持数据块_产品型号", 8); ActivateScreen("欢迎-管理员", 0)
   Button "在线_9" at 488,221 size 100x40; TextOn '在线'; TextOff '备用'
      on Release: SetTag("保持数据块_产品型号", 9); ActivateScreen("欢迎-管理员", 0)
   Button "在线_10" at 626,221 size 100x40; TextOn '在线'; TextOff '备用'
      on Release: SetTag("保持数据块_产品型号", 10); ActivateScreen("欢迎-管理员", 0)
   TextField "文本域_3" at 68,91 size 105x36; Text '当前产品'
   Button "HmiScreenItemData_1" at 71,296 size 103x35; TextOff '用户管理'; PictureOn "Navigates to 用户管理 for KTP900 Basic+ PN 14.0.1.0"; PictureOff "Navigates to 用户管理 for KTP900 Basic+ PN 14.0.1.0"; Authorization "User administration"
      on Release: ActivateScreen("用户管理", 0)
   Button "在线_6" at 73,221 size 100x40; TextOn 'R544'; TextOff 'R567X'
      on Press: function_eba64363(1, U 6, 1, N); function_b431313b(1, U 6, N); ActivateScreen("欢迎-管理员", 0); SetTag("保持数据块_产品型号", 6)

screen "欢迎-管理员" 800x480, template "模板"
   Rectangle "矩形_12" at 686,245 size 97x177
      Appearance <- "后升降台降到位"
   Rectangle "矩形_18" at 686,245 size 63x89
      Appearance <- "后升降台升到位"
   Rectangle "矩形_3" at 226,245 size 97x177
      Appearance <- "前升降台降到位"
   Rectangle "矩形_16" at 260,245 size 63x89
      Appearance <- "前升降台升到位"
   SymbolicIOField "符号 I/O 域_1" at 103,96 size 103x31; TextOn '1'; TextOff '0'; TextList "产品型号"
      ProcessValue <- "保持数据块_产品型号"
   TextField "文本域_3" at 13,97 size 90x28; Text '当前产品：'
   Button "在线_1" at 105,136 size 100x40; TextOn '在线'; TextOff '进入产品选择'
      on Press: ActivateScreen("产品选择", 0)
   TextField "文本域_4" at 76,66 size 73x28; Text '产品信息'
   TextField "文本域_13" at 75,191 size 90x28; Text '传输线控制'
   TextField "文本域_1" at 0,0 size 800x50; Text '主页面'
   Switch "开关_1" at 15,384 size 100x40; TextOn '自动放行'; CaptionText 'Switch'; TextOff '手动放行'
      ProcessValue <- "保持数据块_手动放行/自动放行"
   TextField "文本域_17" at 28,362 size 73x20; Text '放行模式'
   Button "在线_2" at 122,242 size 100x40; TextOn '停止自动'; TextOff '停止'
      on Release: ResetBit("线体停止HMI")
      on Press: SetBit("线体停止HMI")
   TextField "文本域_7" at 127,221 size 90x20; Text '停止传输线'
   Button "在线_3" at 15,242 size 100x40; TextOn '恢复自动'; TextOff '启动'
      on Release: ResetBit("线体启动HMI")
      on Press: SetBit("线体启动HMI")
   TextField "文本域_2" at 20,221 size 90x20; Text '启动传输线'
   Rectangle "矩形_2" at 342,268 size 29x17
      Appearance <- "工位7光电检测"
   Circle "圆_1" at 261,302 size 62x62
      Appearance <- "前升降台皮带电机正在工作"
   Rectangle "矩形_6" at 391,268 size 29x17
      Appearance <- "工位6光电检测"
   Rectangle "矩形_7" at 440,268 size 29x17
      Appearance <- "工位5光电检测"
   Rectangle "矩形_8" at 489,268 size 29x17
      Appearance <- "工位4光电检测"
   Rectangle "矩形_9" at 538,268 size 29x17
      Appearance <- "工位3光电检测"
   Rectangle "矩形_10" at 587,268 size 29x17
      Appearance <- "工位2光电检测"
   Rectangle "矩形_11" at 636,268 size 29x17
      Appearance <- "工位1光电检测"
   Circle "圆_2" at 686,302 size 62x62
      Appearance <- "后升降台皮带电机正在工作"
   Rectangle "矩形_13" at 342,373 size 29x17
      Appearance <- "前方下轨道出料口有料检测"
   Rectangle "矩形_15" at 636,373 size 29x17
      Appearance <- "后方下轨道进料口有料检测"
   TextField "文本域_5" at 631,246 size 41x17; Text '工位1'
   TextField "文本域_6" at 581,246 size 41x17; Text '工位2'
   TextField "文本域_8" at 533,246 size 41x17; Text '工位3'
   TextField "文本域_9" at 483,246 size 41x17; Text '工位4'
   TextField "文本域_10" at 434,246 size 41x17; Text '工位5'
   TextField "文本域_11" at 386,246 size 41x17; Text '工位6'
   TextField "文本域_12" at 336,246 size 41x17; Text '工位7'
   TextField "文本域_14" at 239,221 size 73x20; Text '前升降台'
   TextField "文本域_15" at 698,221 size 73x20; Text '后升降台'
   TextField "文本域_16" at 329,354 size 61x17; Text '出料感应'
   TextField "文本域_18" at 623,354 size 61x17; Text '进料感应'
   Rectangle "矩形_14" at 226,245 size 36x177
      Appearance <- "前升降台有料检测"
   Rectangle "矩形_17" at 747,245 size 36x177
      Appearance <- "后升降台有料检测"
   TextField "文本域_19" at 268,260 size 47x17; Text '升到位'
      Visibility <- "前升降台升到位"
   TextField "文本域_20" at 268,389 size 47x17; Text '降到位'
      Visibility <- "前升降台降到位"
   TextField "文本域_21" at 234,308 size 19x43; Text '有 料'
      Visibility <- "前升降台有料检测"
   TextField "文本域_22" at 234,308 size 19x43; Text '无 料'
      Visibility <- "前升降台有料检测"
   TextField "文本域_23" at 756,307 size 19x43; Text '有 料'
      Visibility <- "后升降台有料检测"
   TextField "文本域_24" at 756,307 size 19x43; Text '无 料'
      Visibility <- "后升降台有料检测"
   TextField "文本域_25" at 694,260 size 47x17; Text '升到位'
      Visibility <- "后升降台升到位"
   TextField "文本域_26" at 695,389 size 47x17; Text '降到位'
      Visibility <- "后升降台降到位"
   SymbolicIOField "符号 I/O 域_3" at 265,320 size 52x26; TextOn '1'; TextOff '0'; TextList "前升降皮带工作状态"
      ProcessValue <- "前升降台皮带电机显示到HMI状态号"
   SymbolicIOField "符号 I/O 域_2" at 690,320 size 52x26; TextOn '1'; TextOff '0'; TextList "后升降皮带工作状态"
      ProcessValue <- "后升降台皮带电机显示到HMI状态号"
   Rectangle "矩形_19" at 322,284 size 109x33
      Appearance <- "前输送线电机显示到HMI状态号"
   Rectangle "矩形_20" at 578,389 size 109x33
      Appearance <- "后输送线电机显示到HMI状态号"
   TextField "文本域_27" at 225,106 size 130x37; Text '设备状态：'
   SymbolicIOField "符号 I/O 域_4" at 348,91 size 418x67; TextOn '1'; TextOff '0'; TextList "设备状态显示"
      ProcessValue <- "设备状态号"
   IOField "I/O 域_1" at 15,316 size 100x40; FormatPattern 99; Unit Hz
      ProcessValue <- "保持数据块_前输送电机变频器设定频率"
   TextField "文本域_28" at 10,292 size 107x20; Text '上传输线速度'
   IOField "I/O 域_2" at 122,316 size 100x40; FormatPattern 99; Unit Hz
      ProcessValue <- "保持数据块_后输送电机变频器设定频率"
   TextField "文本域_29" at 117,292 size 107x20; Text '下传输线速度'
   SymbolicIOField "符号 I/O 域_5" at 326,289 size 97x26; TextOn '1'; TextOff '0'; TextList "上输送线工作状态"
      ProcessValue <- "前输送线电机显示到HMI状态号"
   SymbolicIOField "符号 I/O 域_6" at 584,393 size 97x26; TextOn '1'; TextOff '0'; TextList "下输送线工作状态"
      ProcessValue <- "后输送线电机显示到HMI状态号"
   Button "在线_4" at 121,384 size 100x40; TextOn '停止自动'; TextOff '清除故障'
      on Release: ResetBit("故障复位HMI")
      on Press: SetBit("故障复位HMI")
   TextField "文本域_30" at 134,363 size 73x20; Text '清除故障'
   TextField "文本域_31" at 442,191 size 124x28; Text '传输线工作状态'

Template "模板" 800x480
   GraphicView "模板_图形视图_1" at 0,0 size 800x480; Picture "HMI_BG"
   Button "退出" at 707,442 size 80x35; TextOff '退出'; PictureOn "ExitRuntime_KTP900_Basic_PN_TR"; PictureOff "ExitRuntime_KTP900_Basic_PN_TR"
      on Release: StopRuntime(0)
   Button "Template_Button_1" at 567,442 size 80x35; TextOn 'IO监控'; TextOff 'IO监控'
      on Release: ActivateScreen("DI_1", 0)
   Button "Template_Button_3" at 301,442 size 80x35; TextOn '手动'; TextOff '手动'
      on Release: ActivateScreen("输送线气缸", 0)
   Button "起始画面" at 160,442 size 80x35; TextOff '主页'; PictureOn "NavigateHome_KTP900_Basic_PN_TR"; PictureOff "NavigateHome_KTP900_Basic_PN_TR"
      on Release: ActivateScreen("欢迎-管理员", 0)
   Button "报警" at 18,442 size 80x35; TextOff '报警'; PictureOn "AlarmDisplay_KTP900_Basic_PN_TR"; PictureOff "AlarmDisplay_KTP900_Basic_PN_TR"
      on Release: ActivateScreen("报警画面", 0)
   Button "模板_按钮_1" at 433,442 size 82x38; TextOff '参数设置'
      on Release: ActivateScreen("配方", 0)

Template "登陆" 800x480
   GraphicView "模板_图形视图_1" at 0,0 size 800x480; Picture "HMI_Login"
   IOField "模板_I/O 域_1" at 232,194 size 307x32; FormatPattern ????????????????????????????????????
      ProcessValue <- "用户名"
   IOField "模板_I/O 域_2" at 232,274 size 307x32; FormatPattern ????????????????????????????????????
      ProcessValue <- "密码"
   Button "模板_按钮_1" at 231,330 size 339x39; TextOff '登陆'
      on Release: function_e1ab61de("编号"); ActivateScreenByNumber("编号", 0)
      on Press: function_a9b89908("密码", "用户名")

screen "报警画面" 800x480, template "模板"
   AlarmView "报警视图_1" at 13,65 size 775x365
   TextField "文本域_4" at 0,0 size 800x50; Text '报警画面'

screen "用户管理" 800x480, template "模板"
   UserView "HmiScreenItemData" at 9,61 size 782x371
   TextField "文本域_6" at 0,0 size 800x50; Text '用户管理'

screen "配方" 800x480, template "模板"
   RecipeView "配方视图_1" at 11,62 size 776x368; ValueCaption '设定值'; RecipeNameCaption '设备名称：'; EntryNameCaption '参数名称'; DataRecordNameCaption '产品选择：'; Recipe "传输线参数写入"
   TextField "文本域_2" at 0,0 size 800x50; Text '参数设置'
*)